LIN {X 0,Y 448.566,Z 349.616,A -85,B 0,C 180,E1 -8842.421,E2 -8842.421} C_VEL
LIN {X 0,Y 446.487,Z 338.496,A -85,B 0,C 180,E1 -8844.517,E2 -8844.517} C_VEL
LIN {X 0,Y 446.478,Z 338.493,A -85,B 0,C 180,E1 -8847.161,E2 -8847.161} C_VEL
LIN {X 0,Y 446.433,Z 338.501,A -85,B 0,C 180,E1 -8850.249,E2 -8850.249} C_VEL
LIN {X 0,Y 446.451,Z 338.496,A -85,B 0,C 180,E1 -8853.453,E2 -8853.453} C_VEL
LIN {X 0,Y 446.405,Z 338.501,A -85,B 0,C 180,E1 -8856.745,E2 -8856.745} C_VEL
LIN {X 0,Y 446.406,Z 338.503,A -85,B 0,C 180,E1 -8859.516,E2 -8859.516} C_VEL
LIN {X 0,Y 446.421,Z 338.499,A -85,B 0,C 180,E1 -8862.606,E2 -8862.606} C_VEL
LIN {X 0,Y 446.455,Z 338.496,A -85,B 0,C 180,E1 -8865.103,E2 -8865.103} C_VEL
LIN {X 0,Y 446.411,Z 338.5,A -85,B 0,C 180,E1 -8868.606,E2 -8868.606} C_VEL
LIN {X 0,Y 446.404,Z 338.505,A -85,B 0,C 180,E1 -8871.923,E2 -8871.923} C_VEL
LIN {X 0,Y 446.425,Z 338.501,A -85,B 0,C 180,E1 -8875.475,E2 -8875.475} C_VEL
LIN {X 0,Y 446.394,Z 338.506,A -85,B 0,C 180,E1 -8878.697,E2 -8878.697} C_VEL
LIN {X 0,Y 446.41,Z 338.504,A -85,B 0,C 180,E1 -8881.84,E2 -8881.84} C_VEL
LIN {X 0,Y 446.427,Z 338.66,A -85,B 0,C 180,E1 -8883.514,E2 -8883.514} C_VEL
LIN {X 0,Y 449.208,Z 351.748,A -85,B 0,C 180,E1 -8886.241,E2 -8886.241} C_VEL
LIN {X 0,Y 449.635,Z 355.585,A -85,B 0,C 180,E1 -8887.001,E2 -8887.001} C_VEL
LIN {X 0,Y 449.143,Z 363.301,A -85,B 0,C 180,E1 -8888.438,E2 -8888.438} C_VEL
LIN {X 0,Y 450.701,Z 371.004,A -85,B 0,C 180,E1 -8888.654,E2 -8888.654} C_VEL
LIN {X 0,Y 451.103,Z 376.824,A -85,B 0,C 180,E1 -8888.771,E2 -8888.771} C_VEL
LIN {X 0,Y 450.451,Z 382.718,A -85,B 0,C 180,E1 -8888.837,E2 -8888.837} C_VEL
LIN {X 0,Y 447.177,Z 398.482,A -85,B 0,C 180,E1 -8888.94,E2 -8888.94} C_VEL
LIN {X 0,Y 446.777,Z 402.479,A -85,B 0,C 180,E1 -8888.988,E2 -8888.988} C_VEL
LIN {X 0,Y 445.528,Z 498.742,A -85,B 0,C 180,E1 -8890.563,E2 -8890.563} C_VEL
LIN {X 0,Y 445.071,Z 513.383,A -85,B 0,C 180,E1 -8890.962,E2 -8890.962} C_VEL
LIN {X 0,Y 444.548,Z 526.67,A -85,B 0,C 180,E1 -8891.507,E2 -8891.507} C_VEL
LIN {X 0,Y 443.844,Z 539.571,A -85,B 0,C 180,E1 -8892.212,E2 -8892.212} C_VEL
LIN {X 0,Y 443.131,Z 551.657,A -85,B 0,C 180,E1 -8893.056,E2 -8893.056} C_VEL
LIN {X 0,Y 442.208,Z 563.631,A -85,B 0,C 180,E1 -8894.087,E2 -8894.087} C_VEL
LIN {X 0,Y 441.379,Z 574.55,A -85,B 0,C 180,E1 -8895.239,E2 -8895.239} C_VEL
LIN {X 0,Y 440.642,Z 584.036,A -85,B 0,C 180,E1 -8896.441,E2 -8896.441} C_VEL
LIN {X 0,Y 440.079,Z 592.855,A -85,B 0,C 180,E1 -8897.783,E2 -8897.783} C_VEL
LIN {X 0,Y 439.351,Z 601.602,A -85,B 0,C 180,E1 -8899.398,E2 -8899.398} C_VEL
LIN {X 0,Y 438.986,Z 607.768,A -85,B 0,C 180,E1 -8900.786,E2 -8900.786} C_VEL
LIN {X 0,Y 438.615,Z 614.306,A -85,B 0,C 180,E1 -8902.634,E2 -8902.634} C_VEL
LIN {X 0,Y 438.46,Z 619.203,A -85,B 0,C 180,E1 -8904.48,E2 -8904.48} C_VEL
LIN {X 0,Y 438.291,Z 622.617,A -85,B 0,C 180,E1 -8906.321,E2 -8906.321} C_VEL
LIN {X 0,Y 438.342,Z 623.801,A -85,B 0,C 180,E1 -8907.242,E2 -8907.242} C_VEL
LIN {X 0,Y 438.229,Z 625.165,A -85,B 0,C 180,E1 -8909.08,E2 -8909.08} C_VEL
LIN {X 0,Y 438.229,Z 625.204,A -85,B 0,C 180,E1 -8910.918,E2 -8910.918} C_VEL
LIN {X 0,Y 438.34,Z 623.919,A -85,B 0,C 180,E1 -8912.756,E2 -8912.756} C_VEL
LIN {X 0,Y 438.35,Z 621.277,A -85,B 0,C 180,E1 -8914.597,E2 -8914.597} C_VEL
LIN {X 0,Y 438.505,Z 617.205,A -85,B 0,C 180,E1 -8916.44,E2 -8916.44} C_VEL
LIN {X 0,Y 438.771,Z 611.583,A -85,B 0,C 180,E1 -8918.287,E2 -8918.287} C_VEL
LIN {X 0,Y 439.168,Z 605.239,A -85,B 0,C 180,E1 -8919.904,E2 -8919.904} C_VEL
LIN {X 0,Y 439.724,Z 597.348,A -85,B 0,C 180,E1 -8921.523,E2 -8921.523} C_VEL
LIN {X 0,Y 440.33,Z 588.346,A -85,B 0,C 180,E1 -8923.029,E2 -8923.029} C_VEL
LIN {X 0,Y 441.022,Z 579.149,A -85,B 0,C 180,E1 -8924.299,E2 -8924.299} C_VEL
LIN {X 0,Y 441.871,Z 568.079,A -85,B 0,C 180,E1 -8925.567,E2 -8925.567} C_VEL
LIN {X 0,Y 442.7,Z 557.061,A -85,B 0,C 180,E1 -8926.602,E2 -8926.602} C_VEL
LIN {X 0,Y 443.617,Z 543.849,A -85,B 0,C 180,E1 -8927.602,E2 -8927.602} C_VEL
LIN {X 0,Y 444.29,Z 531.223,A -85,B 0,C 180,E1 -8928.357,E2 -8928.357} C_VEL
LIN {X 0,Y 444.92,Z 517.384,A -85,B 0,C 180,E1 -8928.982,E2 -8928.982} C_VEL
LIN {X 0,Y 445.448,Z 502.754,A -85,B 0,C 180,E1 -8929.437,E2 -8929.437} C_VEL
LIN {X 0,Y 445.804,Z 478.658,A -85,B 0,C 180,E1 -8929.871,E2 -8929.871} C_VEL
LIN {X 0,Y 446.948,Z 386.866,A -85,B 0,C 180,E1 -8931.362,E2 -8931.362} C_VEL
LIN {X 0,Y 443.134,Z 367.334,A -85,B 0,C 180,E1 -8931.889,E2 -8931.889} C_VEL
LIN {X 0,Y 442.319,Z 363.353,A -85,B 0,C 180,E1 -8932.01,E2 -8932.01} C_VEL
LIN {X 0,Y 442.779,Z 356.138,A -85,B 0,C 180,E1 -8933.377,E2 -8933.377} C_VEL
LIN {X 0,Y 440.804,Z 345.968,A -85,B 0,C 180,E1 -8935.496,E2 -8935.496} C_VEL
LIN {X 0,Y 439.369,Z 339.384,A -85,B 0,C 180,E1 -8936.927,E2 -8936.927} C_VEL
LIN {X 0,Y 439.367,Z 339.383,A -85,B 0,C 180,E1 -8940.257,E2 -8940.257} C_VEL
LIN {X 0,Y 439.389,Z 339.379,A -85,B 0,C 180,E1 -8943.722,E2 -8943.722} C_VEL
LIN {X 0,Y 439.337,Z 339.389,A -85,B 0,C 180,E1 -8946.885,E2 -8946.885} C_VEL
LIN {X 0,Y 439.337,Z 339.382,A -85,B 0,C 180,E1 -8949.839,E2 -8949.839} C_VEL
LIN {X 0,Y 439.323,Z 339.387,A -85,B 0,C 180,E1 -8952.618,E2 -8952.618} C_VEL
LIN {X 0,Y 439.387,Z 339.377,A -85,B 0,C 180,E1 -8955.269,E2 -8955.269} C_VEL
LIN {X 0,Y 439.344,Z 339.386,A -85,B 0,C 180,E1 -8959.015,E2 -8959.015} C_VEL
LIN {X 0,Y 439.333,Z 339.378,A -85,B 0,C 180,E1 -8962.563,E2 -8962.563} C_VEL
LIN {X 0,Y 439.383,Z 339.381,A -85,B 0,C 180,E1 -8964.842,E2 -8964.842} C_VEL
LIN {X 0,Y 439.353,Z 339.372,A -85,B 0,C 180,E1 -8968.138,E2 -8968.138} C_VEL
LIN {X 0,Y 439.386,Z 339.372,A -85,B 0,C 180,E1 -8971.605,E2 -8971.605} C_VEL
LIN {X 0,Y 439.356,Z 339.37,A -85,B 0,C 180,E1 -8974.412,E2 -8974.412} C_VEL
LIN {X 0,Y 439.349,Z 339.38,A -85,B 0,C 180,E1 -8977.424,E2 -8977.424} C_VEL
LIN {X 0,Y 439.427,Z 339.36,A -85,B 0,C 180,E1 -8980.663,E2 -8980.663} C_VEL
LIN {X 0,Y 439.439,Z 339.369,A -85,B 0,C 180,E1 -8984.224,E2 -8984.224} C_VEL
LIN {X 0,Y 439.467,Z 339.364,A -85,B 0,C 180,E1 -8988.001,E2 -8988.001} C_VEL
LIN {X 0,Y 439.487,Z 339.359,A -85,B 0,C 180,E1 -8991.725,E2 -8991.725} C_VEL
LIN {X 0,Y 439.575,Z 339.355,A -85,B 0,C 180,E1 -8994.495,E2 -8994.495} C_VEL
LIN {X 0,Y 439.615,Z 339.349,A -85,B 0,C 180,E1 -8998.168,E2 -8998.168} C_VEL
LIN {X 0,Y 439.58,Z 339.354,A -85,B 0,C 180,E1 -9000.916,E2 -9000.916} C_VEL
LIN {X 0,Y 439.594,Z 339.352,A -85,B 0,C 180,E1 -9002.749,E2 -9002.749} C_VEL
LIN {X 0,Y 439.546,Z 339.361,A -85,B 0,C 180,E1 -9006.426,E2 -9006.426} C_VEL
LIN {X 0,Y 439.459,Z 339.365,A -85,B 0,C 180,E1 -9009.202,E2 -9009.202} C_VEL
LIN {X 0,Y 439.45,Z 339.367,A -85,B 0,C 180,E1 -9012.938,E2 -9012.938} C_VEL
LIN {X 0,Y 439.431,Z 339.373,A -85,B 0,C 180,E1 -9016.348,E2 -9016.348} C_VEL
LIN {X 0,Y 439.387,Z 339.374,A -85,B 0,C 180,E1 -9019.627,E2 -9019.627} C_VEL
LIN {X 0,Y 439.347,Z 339.372,A -85,B 0,C 180,E1 -9022.576,E2 -9022.576} C_VEL
LIN {X 0,Y 439.35,Z 339.379,A -85,B 0,C 180,E1 -9025.588,E2 -9025.588} C_VEL
LIN {X 0,Y 439.376,Z 339.369,A -85,B 0,C 180,E1 -9028.676,E2 -9028.676} C_VEL
LIN {X 0,Y 439.349,Z 339.383,A -85,B 0,C 180,E1 -9032.03,E2 -9032.03} C_VEL
LIN {X 0,Y 439.373,Z 339.376,A -85,B 0,C 180,E1 -9035.34,E2 -9035.34} C_VEL
LIN {X 0,Y 439.338,Z 339.385,A -85,B 0,C 180,E1 -9038.6,E2 -9038.6} C_VEL
LIN {X 0,Y 439.347,Z 339.379,A -85,B 0,C 180,E1 -9041.253,E2 -9041.253} C_VEL
LIN {X 0,Y 439.363,Z 339.381,A -85,B 0,C 180,E1 -9044.734,E2 -9044.734} C_VEL
LIN {X 0,Y 439.334,Z 339.386,A -85,B 0,C 180,E1 -9047.791,E2 -9047.791} C_VEL
LIN {X 0,Y 439.339,Z 339.383,A -85,B 0,C 180,E1 -9051.403,E2 -9051.403} C_VEL
LIN {X 0,Y 439.382,Z 339.378,A -85,B 0,C 180,E1 -9054.845,E2 -9054.845} C_VEL
LIN {X 0,Y 439.358,Z 339.383,A -85,B 0,C 180,E1 -9058.14,E2 -9058.14} C_VEL
LIN {X 0,Y 439.38,Z 339.378,A -85,B 0,C 180,E1 -9061.611,E2 -9061.611} C_VEL
LIN {X 0,Y 439.386,Z 339.457,A -85,B 0,C 180,E1 -9061.961,E2 -9061.961} C_VEL
LIN {X 0,Y 442.5,Z 353.697,A -85,B 0,C 180,E1 -9064.864,E2 -9064.864} C_VEL
LIN {X 0,Y 443.085,Z 357.713,A -85,B 0,C 180,E1 -9065.646,E2 -9065.646} C_VEL
LIN {X 0,Y 442.195,Z 370.912,A -85,B 0,C 180,E1 -9068.034,E2 -9068.034} C_VEL
LIN {X 0,Y 446.887,Z 395.742,A -85,B 0,C 180,E1 -9068.697,E2 -9068.697} C_VEL
LIN {X 0,Y 445.457,Z 507.784,A -85,B 0,C 180,E1 -9070.533,E2 -9070.533} C_VEL
LIN {X 0,Y 444.963,Z 521.924,A -85,B 0,C 180,E1 -9070.93,E2 -9070.93} C_VEL
LIN {X 0,Y 444.358,Z 535.626,A -85,B 0,C 180,E1 -9071.501,E2 -9071.501} C_VEL
LIN {X 0,Y 443.601,Z 549.079,A -85,B 0,C 180,E1 -9072.255,E2 -9072.255} C_VEL
LIN {X 0,Y 442.82,Z 561.734,A -85,B 0,C 180,E1 -9073.165,E2 -9073.165} C_VEL
LIN {X 0,Y 441.889,Z 573.37,A -85,B 0,C 180,E1 -9074.197,E2 -9074.197} C_VEL
LIN {X 0,Y 441.181,Z 583.057,A -85,B 0,C 180,E1 -9075.235,E2 -9075.235} C_VEL
LIN {X 0,Y 440.395,Z 593.68,A -85,B 0,C 180,E1 -9076.606,E2 -9076.606} C_VEL
LIN {X 0,Y 439.801,Z 602.653,A -85,B 0,C 180,E1 -9078.012,E2 -9078.012} C_VEL
LIN {X 0,Y 439.143,Z 611.145,A -85,B 0,C 180,E1 -9079.629,E2 -9079.629} C_VEL
LIN {X 0,Y 438.778,Z 617.986,A -85,B 0,C 180,E1 -9081.249,E2 -9081.249} C_VEL
LIN {X 0,Y 438.515,Z 622.7,A -85,B 0,C 180,E1 -9082.635,E2 -9082.635} C_VEL
LIN {X 0,Y 438.423,Z 627.591,A -85,B 0,C 180,E1 -9084.482,E2 -9084.482} C_VEL
LIN {X 0,Y 438.25,Z 630.988,A -85,B 0,C 180,E1 -9086.324,E2 -9086.324} C_VEL
LIN {X 0,Y 438.27,Z 632.994,A -85,B 0,C 180,E1 -9088.164,E2 -9088.164} C_VEL
LIN {X 0,Y 438.227,Z 633.656,A -85,B 0,C 180,E1 -9090.001,E2 -9090.001} C_VEL
LIN {X 0,Y 438.271,Z 632.988,A -85,B 0,C 180,E1 -9091.839,E2 -9091.839} C_VEL
LIN {X 0,Y 438.25,Z 630.975,A -85,B 0,C 180,E1 -9093.679,E2 -9093.679} C_VEL
LIN {X 0,Y 438.396,Z 627.576,A -85,B 0,C 180,E1 -9095.521,E2 -9095.521} C_VEL
LIN {X 0,Y 438.517,Z 622.686,A -85,B 0,C 180,E1 -9097.368,E2 -9097.368} C_VEL
LIN {X 0,Y 438.87,Z 616.152,A -85,B 0,C 180,E1 -9099.216,E2 -9099.216} C_VEL
LIN {X 0,Y 439.301,Z 608.881,A -85,B 0,C 180,E1 -9100.836,E2 -9100.836} C_VEL
LIN {X 0,Y 440.002,Z 599.879,A -85,B 0,C 180,E1 -9102.454,E2 -9102.454} C_VEL
LIN {X 0,Y 440.623,Z 590.428,A -85,B 0,C 180,E1 -9103.844,E2 -9103.844} C_VEL
LIN {X 0,Y 441.423,Z 579.967,A -85,B 0,C 180,E1 -9105.113,E2 -9105.113} C_VEL
LIN {X 0,Y 442.283,Z 568.419,A -85,B 0,C 180,E1 -9106.265,E2 -9106.265} C_VEL
LIN {X 0,Y 443.191,Z 555.607,A -85,B 0,C 180,E1 -9107.299,E2 -9107.299} C_VEL
LIN {X 0,Y 444.049,Z 542.285,A -85,B 0,C 180,E1 -9108.146,E2 -9108.146} C_VEL
LIN {X 0,Y 444.642,Z 529.175,A -85,B 0,C 180,E1 -9108.788,E2 -9108.788} C_VEL
LIN {X 0,Y 445.256,Z 515.429,A -85,B 0,C 180,E1 -9109.269,E2 -9109.269} C_VEL
LIN {X 0,Y 445.561,Z 501.404,A -85,B 0,C 180,E1 -9109.585,E2 -9109.585} C_VEL
LIN {X 0,Y 446.869,Z 395.827,A -85,B 0,C 180,E1 -9111.298,E2 -9111.298} C_VEL
LIN {X 0,Y 442.566,Z 372.827,A -85,B 0,C 180,E1 -9111.908,E2 -9111.908} C_VEL
LIN {X 0,Y 442.209,Z 370.731,A -85,B 0,C 180,E1 -9111.994,E2 -9111.994} C_VEL
LIN {X 0,Y 443.057,Z 357.667,A -85,B 0,C 180,E1 -9114.358,E2 -9114.358} C_VEL
LIN {X 0,Y 441.922,Z 350.934,A -85,B 0,C 180,E1 -9115.682,E2 -9115.682} C_VEL
LIN {X 0,Y 439.383,Z 339.381,A -85,B 0,C 180,E1 -9118.071,E2 -9118.071} C_VEL
LIN {X 0,Y 439.364,Z 339.382,A -85,B 0,C 180,E1 -9120.789,E2 -9120.789} C_VEL
LIN {X 0,Y 439.392,Z 339.377,A -85,B 0,C 180,E1 -9124.044,E2 -9124.044} C_VEL
LIN {X 0,Y 439.351,Z 339.381,A -85,B 0,C 180,E1 -9126.887,E2 -9126.887} C_VEL
LIN {X 0,Y 439.407,Z 339.372,A -85,B 0,C 180,E1 -9129.85,E2 -9129.85} C_VEL
LIN {X 0,Y 439.387,Z 339.377,A -85,B 0,C 180,E1 -9132.628,E2 -9132.628} C_VEL
LIN {X 0,Y 439.407,Z 339.376,A -85,B 0,C 180,E1 -9135.271,E2 -9135.271} C_VEL
LIN {X 0,Y 439.394,Z 339.378,A -85,B 0,C 180,E1 -9138.744,E2 -9138.744} C_VEL
LIN {X 0,Y 439.381,Z 339.377,A -85,B 0,C 180,E1 -9141.608,E2 -9141.608} C_VEL
LIN {X 0,Y 439.403,Z 339.375,A -85,B 0,C 180,E1 -9144.844,E2 -9144.844} C_VEL
LIN {X 0,Y 439.378,Z 339.382,A -85,B 0,C 180,E1 -9148.14,E2 -9148.14} C_VEL
LIN {X 0,Y 439.413,Z 339.381,A -85,B 0,C 180,E1 -9151.604,E2 -9151.604} C_VEL
LIN {X 0,Y 439.396,Z 339.439,A -85,B 0,C 180,E1 -9154.542,E2 -9154.542} C_VEL
LIN {X 0,Y 442.118,Z 350.97,A -85,B 0,C 180,E1 -9156.77,E2 -9156.77} C_VEL
LIN {X 0,Y 442.617,Z 355.527,A -85,B 0,C 180,E1 -9157.599,E2 -9157.599} C_VEL
LIN {X 0,Y 442.149,Z 372.27,A -85,B 0,C 180,E1 -9160.501,E2 -9160.501} C_VEL
LIN {X 0,Y 441.97,Z 378.87,A -85,B 0,C 180,E1 -9161.636,E2 -9161.636} C_VEL
LIN {X 0,Y 444.896,Z 393.264,A -85,B 0,C 180,E1 -9162.133,E2 -9162.133} C_VEL
LIN {X 0,Y 443.215,Z 477.735,A -85,B 0,C 180,E1 -9163.86,E2 -9163.86} C_VEL
LIN {X 0,Y 442.985,Z 491.998,A -85,B 0,C 180,E1 -9164.206,E2 -9164.206} C_VEL
LIN {X 0,Y 442.582,Z 504.819,A -85,B 0,C 180,E1 -9164.693,E2 -9164.693} C_VEL
LIN {X 0,Y 442.177,Z 515.784,A -85,B 0,C 180,E1 -9165.268,E2 -9165.268} C_VEL
LIN {X 0,Y 441.569,Z 528.484,A -85,B 0,C 180,E1 -9166.14,E2 -9166.14} C_VEL
LIN {X 0,Y 441.069,Z 539.531,A -85,B 0,C 180,E1 -9167.11,E2 -9167.11} C_VEL
LIN {X 0,Y 440.43,Z 550.006,A -85,B 0,C 180,E1 -9168.261,E2 -9168.261} C_VEL
LIN {X 0,Y 439.96,Z 558.544,A -85,B 0,C 180,E1 -9169.415,E2 -9169.415} C_VEL
LIN {X 0,Y 439.464,Z 566.835,A -85,B 0,C 180,E1 -9170.798,E2 -9170.798} C_VEL
LIN {X 0,Y 439.078,Z 573.477,A -85,B 0,C 180,E1 -9172.181,E2 -9172.181} C_VEL
LIN {X 0,Y 438.888,Z 578.742,A -85,B 0,C 180,E1 -9173.564,E2 -9173.564} C_VEL
LIN {X 0,Y 438.541,Z 582.812,A -85,B 0,C 180,E1 -9174.943,E2 -9174.943} C_VEL
LIN {X 0,Y 438.57,Z 585.775,A -85,B 0,C 180,E1 -9176.325,E2 -9176.325} C_VEL
LIN {X 0,Y 438.45,Z 587.197,A -85,B 0,C 180,E1 -9177.244,E2 -9177.244} C_VEL
LIN {X 0,Y 438.376,Z 588.173,A -85,B 0,C 180,E1 -9178.163,E2 -9178.163} C_VEL
LIN {X 0,Y 438.339,Z 588.748,A -85,B 0,C 180,E1 -9179.081,E2 -9179.081} C_VEL
LIN {X 0,Y 438.313,Z 588.9,A -85,B 0,C 180,E1 -9180,E2 -9180} C_VEL
LIN {X 0,Y 438.31,Z 588.599,A -85,B 0,C 180,E1 -9180.919,E2 -9180.919} C_VEL
LIN {X 0,Y 438.35,Z 587.898,A -85,B 0,C 180,E1 -9181.838,E2 -9181.838} C_VEL
LIN {X 0,Y 438.434,Z 586.788,A -85,B 0,C 180,E1 -9182.756,E2 -9182.756} C_VEL
LIN {X 0,Y 438.488,Z 584.28,A -85,B 0,C 180,E1 -9184.136,E2 -9184.136} C_VEL
LIN {X 0,Y 438.609,Z 580.731,A -85,B 0,C 180,E1 -9185.517,E2 -9185.517} C_VEL
LIN {X 0,Y 438.805,Z 575.437,A -85,B 0,C 180,E1 -9187.05,E2 -9187.05} C_VEL
LIN {X 0,Y 439.08,Z 568.932,A -85,B 0,C 180,E1 -9188.514,E2 -9188.514} C_VEL
LIN {X 0,Y 439.476,Z 561.185,A -85,B 0,C 180,E1 -9189.899,E2 -9189.899} C_VEL
LIN {X 0,Y 439.947,Z 551.471,A -85,B 0,C 180,E1 -9191.285,E2 -9191.285} C_VEL
LIN {X 0,Y 440.502,Z 541.396,A -85,B 0,C 180,E1 -9192.438,E2 -9192.438} C_VEL
LIN {X 0,Y 440.946,Z 530.681,A -85,B 0,C 180,E1 -9193.43,E2 -9193.43} C_VEL
LIN {X 0,Y 441.471,Z 519.08,A -85,B 0,C 180,E1 -9194.286,E2 -9194.286} C_VEL
LIN {X 0,Y 441.878,Z 506.81,A -85,B 0,C 180,E1 -9194.978,E2 -9194.978} C_VEL
LIN {X 0,Y 442.331,Z 493.591,A -85,B 0,C 180,E1 -9195.523,E2 -9195.523} C_VEL
LIN {X 0,Y 442.547,Z 480.562,A -85,B 0,C 180,E1 -9195.87,E2 -9195.87} C_VEL
LIN {X 0,Y 443.737,Z 392.63,A -85,B 0,C 180,E1 -9197.521,E2 -9197.521} C_VEL
LIN {X 0,Y 440.953,Z 376.477,A -85,B 0,C 180,E1 -9197.951,E2 -9197.951} C_VEL
LIN {X 0,Y 441.505,Z 358.045,A -85,B 0,C 180,E1 -9201.232,E2 -9201.232} C_VEL
LIN {X 0,Y 441.535,Z 350.426,A -85,B 0,C 180,E1 -9202.6,E2 -9202.6} C_VEL
LIN {X 0,Y 439.461,Z 339.371,A -85,B 0,C 180,E1 -9204.727,E2 -9204.727} C_VEL
LIN {X 0,Y 439.446,Z 339.371,A -85,B 0,C 180,E1 -9207.632,E2 -9207.632} C_VEL
LIN {X 0,Y 439.367,Z 339.376,A -85,B 0,C 180,E1 -9210.788,E2 -9210.788} C_VEL
LIN {X 0,Y 439.393,Z 339.379,A -85,B 0,C 180,E1 -9214.043,E2 -9214.043} C_VEL
LIN {X 0,Y 439.352,Z 339.38,A -85,B 0,C 180,E1 -9216.886,E2 -9216.886} C_VEL
LIN {X 0,Y 439.353,Z 339.386,A -85,B 0,C 180,E1 -9219.84,E2 -9219.84} C_VEL
LIN {X 0,Y 439.375,Z 339.377,A -85,B 0,C 180,E1 -9222.625,E2 -9222.625} C_VEL
LIN {X 0,Y 439.403,Z 339.376,A -85,B 0,C 180,E1 -9225.27,E2 -9225.27} C_VEL
LIN {X 0,Y 439.362,Z 339.38,A -85,B 0,C 180,E1 -9229.016,E2 -9229.016} C_VEL
LIN {X 0,Y 439.342,Z 339.382,A -85,B 0,C 180,E1 -9232.563,E2 -9232.563} C_VEL
LIN {X 0,Y 439.398,Z 339.376,A -85,B 0,C 180,E1 -9234.843,E2 -9234.843} C_VEL
LIN {X 0,Y 439.35,Z 339.383,A -85,B 0,C 180,E1 -9238.137,E2 -9238.137} C_VEL
LIN {X 0,Y 439.384,Z 339.382,A -85,B 0,C 180,E1 -9241.323,E2 -9241.323} C_VEL
LIN {X 0,Y 439.357,Z 339.437,A -85,B 0,C 180,E1 -9243.198,E2 -9243.198} C_VEL
LIN {X 0,Y 442.298,Z 353.087,A -85,B 0,C 180,E1 -9246.096,E2 -9246.096} C_VEL
LIN {X 0,Y 442.73,Z 357.158,A -85,B 0,C 180,E1 -9246.913,E2 -9246.913} C_VEL
LIN {X 0,Y 442.302,Z 363.377,A -85,B 0,C 180,E1 -9248.088,E2 -9248.088} C_VEL
LIN {X 0,Y 446.951,Z 386.317,A -85,B 0,C 180,E1 -9248.724,E2 -9248.724} C_VEL
LIN {X 0,Y 446.777,Z 402.479,A -85,B 0,C 180,E1 -9248.988,E2 -9248.988} C_VEL
LIN {X 0,Y 445.959,Z 408.324,A -85,B 0,C 180,E1 -9249.046,E2 -9249.046} C_VEL
LIN {X 0,Y 440.489,Z 427.373,A -85,B 0,C 180,E1 -9249.098,E2 -9249.098} C_VEL
LIN {X 0,Y 439.78,Z 433.216,A -85,B 0,C 180,E1 -9249.163,E2 -9249.163} C_VEL
LIN {X 0,Y 438.804,Z 500.275,A -85,B 0,C 180,E1 -9250.284,E2 -9250.284} C_VEL
LIN {X 0,Y 438.287,Z 515.011,A -85,B 0,C 180,E1 -9250.716,E2 -9250.716} C_VEL
LIN {X 0,Y 437.748,Z 527.879,A -85,B 0,C 180,E1 -9251.269,E2 -9251.269} C_VEL
LIN {X 0,Y 436.984,Z 541.227,A -85,B 0,C 180,E1 -9252.032,E2 -9252.032} C_VEL
LIN {X 0,Y 436.234,Z 553.154,A -85,B 0,C 180,E1 -9252.9,E2 -9252.9} C_VEL
LIN {X 0,Y 435.276,Z 564.875,A -85,B 0,C 180,E1 -9253.947,E2 -9253.947} C_VEL
LIN {X 0,Y 434.294,Z 576.569,A -85,B 0,C 180,E1 -9255.233,E2 -9255.233} C_VEL
LIN {X 0,Y 433.505,Z 586.646,A -85,B 0,C 180,E1 -9256.588,E2 -9256.588} C_VEL
LIN {X 0,Y 432.885,Z 595.628,A -85,B 0,C 180,E1 -9258.052,E2 -9258.052} C_VEL
LIN {X 0,Y 432.254,Z 603.886,A -85,B 0,C 180,E1 -9259.696,E2 -9259.696} C_VEL
LIN {X 0,Y 431.837,Z 609.642,A -85,B 0,C 180,E1 -9261.105,E2 -9261.105} C_VEL
LIN {X 0,Y 431.545,Z 614.375,A -85,B 0,C 180,E1 -9262.513,E2 -9262.513} C_VEL
LIN {X 0,Y 431.381,Z 619.272,A -85,B 0,C 180,E1 -9264.389,E2 -9264.389} C_VEL
LIN {X 0,Y 431.197,Z 622.685,A -85,B 0,C 180,E1 -9266.261,E2 -9266.261} C_VEL
LIN {X 0,Y 431.202,Z 624.716,A -85,B 0,C 180,E1 -9268.131,E2 -9268.131} C_VEL
LIN {X 0,Y 431.143,Z 625.417,A -85,B 0,C 180,E1 -9269.999,E2 -9269.999} C_VEL
LIN {X 0,Y 431.201,Z 624.795,A -85,B 0,C 180,E1 -9271.867,E2 -9271.867} C_VEL
LIN {X 0,Y 431.196,Z 622.837,A -85,B 0,C 180,E1 -9273.737,E2 -9273.737} C_VEL
LIN {X 0,Y 431.38,Z 619.492,A -85,B 0,C 180,E1 -9275.608,E2 -9275.608} C_VEL
LIN {X 0,Y 431.541,Z 614.663,A -85,B 0,C 180,E1 -9277.485,E2 -9277.485} C_VEL
LIN {X 0,Y 431.945,Z 608.204,A -85,B 0,C 180,E1 -9279.362,E2 -9279.362} C_VEL
LIN {X 0,Y 432.399,Z 601.013,A -85,B 0,C 180,E1 -9281.008,E2 -9281.008} C_VEL
LIN {X 0,Y 433.075,Z 593.473,A -85,B 0,C 180,E1 -9282.415,E2 -9282.415} C_VEL
LIN {X 0,Y 433.748,Z 583.935,A -85,B 0,C 180,E1 -9283.898,E2 -9283.898} C_VEL
LIN {X 0,Y 434.607,Z 573.457,A -85,B 0,C 180,E1 -9285.233,E2 -9285.233} C_VEL
LIN {X 0,Y 435.51,Z 562.281,A -85,B 0,C 180,E1 -9286.402,E2 -9286.402} C_VEL
LIN {X 0,Y 436.462,Z 549.915,A -85,B 0,C 180,E1 -9287.45,E2 -9287.45} C_VEL
LIN {X 0,Y 437.224,Z 537.403,A -85,B 0,C 180,E1 -9288.302,E2 -9288.302} C_VEL
LIN {X 0,Y 437.952,Z 523.666,A -85,B 0,C 180,E1 -9289.022,E2 -9289.022} C_VEL
LIN {X 0,Y 438.544,Z 509.091,A -85,B 0,C 180,E1 -9289.573,E2 -9289.573} C_VEL
LIN {X 0,Y 438.986,Z 494.622,A -85,B 0,C 180,E1 -9289.918,E2 -9289.918} C_VEL
LIN {X 0,Y 440.33,Z 387.141,A -85,B 0,C 180,E1 -9291.695,E2 -9291.695} C_VEL
LIN {X 0,Y 435.477,Z 363.381,A -85,B 0,C 180,E1 -9292.382,E2 -9292.382} C_VEL
LIN {X 0,Y 435.821,Z 358.176,A -85,B 0,C 180,E1 -9293.384,E2 -9293.384} C_VEL
LIN {X 0,Y 434.965,Z 352.386,A -85,B 0,C 180,E1 -9294.584,E2 -9294.584} C_VEL
LIN {X 0,Y 432.322,Z 340.261,A -85,B 0,C 180,E1 -9297.238,E2 -9297.238} C_VEL
LIN {X 0,Y 432.335,Z 340.26,A -85,B 0,C 180,E1 -9300.507,E2 -9300.507} C_VEL
LIN {X 0,Y 432.351,Z 340.256,A -85,B 0,C 180,E1 -9304.001,E2 -9304.001} C_VEL
LIN {X 0,Y 432.311,Z 340.261,A -85,B 0,C 180,E1 -9307.195,E2 -9307.195} C_VEL
LIN {X 0,Y 432.279,Z 340.262,A -85,B 0,C 180,E1 -9310.17,E2 -9310.17} C_VEL
LIN {X 0,Y 432.293,Z 340.264,A -85,B 0,C 180,E1 -9313.061,E2 -9313.061} C_VEL
LIN {X 0,Y 432.323,Z 340.255,A -85,B 0,C 180,E1 -9315.663,E2 -9315.663} C_VEL
LIN {X 0,Y 432.298,Z 340.26,A -85,B 0,C 180,E1 -9318.4,E2 -9318.4} C_VEL
LIN {X 0,Y 432.318,Z 340.248,A -85,B 0,C 180,E1 -9321.848,E2 -9321.848} C_VEL
LIN {X 0,Y 432.315,Z 340.255,A -85,B 0,C 180,E1 -9325.32,E2 -9325.32} C_VEL
LIN {X 0,Y 432.303,Z 340.255,A -85,B 0,C 180,E1 -9328.652,E2 -9328.652} C_VEL
LIN {X 0,Y 432.314,Z 340.253,A -85,B 0,C 180,E1 -9331.872,E2 -9331.872} C_VEL
LIN {X 0,Y 432.339,Z 340.251,A -85,B 0,C 180,E1 -9335.545,E2 -9335.545} C_VEL
LIN {X 0,Y 432.335,Z 340.248,A -85,B 0,C 180,E1 -9339.045,E2 -9339.045} C_VEL
LIN {X 0,Y 432.343,Z 340.242,A -85,B 0,C 180,E1 -9342.01,E2 -9342.01} C_VEL
LIN {X 0,Y 432.371,Z 340.252,A -85,B 0,C 180,E1 -9344.925,E2 -9344.925} C_VEL
LIN {X 0,Y 432.443,Z 340.238,A -85,B 0,C 180,E1 -9347.803,E2 -9347.803} C_VEL
LIN {X 0,Y 432.448,Z 340.236,A -85,B 0,C 180,E1 -9351.589,E2 -9351.589} C_VEL
LIN {X 0,Y 432.53,Z 340.234,A -85,B 0,C 180,E1 -9354.405,E2 -9354.405} C_VEL
LIN {X 0,Y 432.584,Z 340.225,A -85,B 0,C 180,E1 -9358.138,E2 -9358.138} C_VEL
LIN {X 0,Y 432.54,Z 340.23,A -85,B 0,C 180,E1 -9360.931,E2 -9360.931} C_VEL
LIN {X 0,Y 432.547,Z 340.229,A -85,B 0,C 180,E1 -9362.794,E2 -9362.794} C_VEL
LIN {X 0,Y 432.56,Z 340.224,A -85,B 0,C 180,E1 -9365.594,E2 -9365.594} C_VEL
LIN {X 0,Y 432.43,Z 340.243,A -85,B 0,C 180,E1 -9368.411,E2 -9368.411} C_VEL
LIN {X 0,Y 432.438,Z 340.244,A -85,B 0,C 180,E1 -9372.197,E2 -9372.197} C_VEL
LIN {X 0,Y 432.415,Z 340.245,A -85,B 0,C 180,E1 -9376.039,E2 -9376.039} C_VEL
LIN {X 0,Y 432.372,Z 340.248,A -85,B 0,C 180,E1 -9379.485,E2 -9379.485} C_VEL
LIN {X 0,Y 432.295,Z 340.252,A -85,B 0,C 180,E1 -9382.966,E2 -9382.966} C_VEL
LIN {X 0,Y 432.303,Z 340.26,A -85,B 0,C 180,E1 -9386.036,E2 -9386.036} C_VEL
LIN {X 0,Y 432.312,Z 340.247,A -85,B 0,C 180,E1 -9389.19,E2 -9389.19} C_VEL
LIN {X 0,Y 432.307,Z 340.26,A -85,B 0,C 180,E1 -9392.444,E2 -9392.444} C_VEL
LIN {X 0,Y 432.319,Z 340.257,A -85,B 0,C 180,E1 -9395.82,E2 -9395.82} C_VEL
LIN {X 0,Y 432.286,Z 340.26,A -85,B 0,C 180,E1 -9399.35,E2 -9399.35} C_VEL
LIN {X 0,Y 432.288,Z 340.26,A -85,B 0,C 180,E1 -9401.802,E2 -9401.802} C_VEL
LIN {X 0,Y 432.321,Z 340.263,A -85,B 0,C 180,E1 -9404.349,E2 -9404.349} C_VEL
LIN {X 0,Y 432.29,Z 340.261,A -85,B 0,C 180,E1 -9407.02,E2 -9407.02} C_VEL
LIN {X 0,Y 432.277,Z 340.266,A -85,B 0,C 180,E1 -9409.83,E2 -9409.83} C_VEL
LIN {X 0,Y 432.286,Z 340.262,A -85,B 0,C 180,E1 -9413.022,E2 -9413.022} C_VEL
LIN {X 0,Y 432.324,Z 340.261,A -85,B 0,C 180,E1 -9416.004,E2 -9416.004} C_VEL
LIN {X 0,Y 432.334,Z 340.255,A -85,B 0,C 180,E1 -9419.493,E2 -9419.493} C_VEL
LIN {X 0,Y 432.377,Z 340.426,A -85,B 0,C 180,E1 -9421.668,E2 -9421.668} C_VEL
LIN {X 0,Y 435.506,Z 354.776,A -85,B 0,C 180,E1 -9424.649,E2 -9424.649} C_VEL
LIN {X 0,Y 436.202,Z 358.993,A -85,B 0,C 180,E1 -9425.49,E2 -9425.49} C_VEL
LIN {X 0,Y 435.394,Z 370.89,A -85,B 0,C 180,E1 -9427.674,E2 -9427.674} C_VEL
LIN {X 0,Y 440.276,Z 396.519,A -85,B 0,C 180,E1 -9428.375,E2 -9428.375} C_VEL
LIN {X 0,Y 438.769,Z 507.731,A -85,B 0,C 180,E1 -9430.224,E2 -9430.224} C_VEL
LIN {X 0,Y 438.254,Z 521.864,A -85,B 0,C 180,E1 -9430.627,E2 -9430.627} C_VEL
LIN {X 0,Y 437.624,Z 535.564,A -85,B 0,C 180,E1 -9431.206,E2 -9431.206} C_VEL
LIN {X 0,Y 436.811,Z 549.336,A -85,B 0,C 180,E1 -9431.992,E2 -9431.992} C_VEL
LIN {X 0,Y 436.011,Z 561.67,A -85,B 0,C 180,E1 -9432.894,E2 -9432.894} C_VEL
LIN {X 0,Y 435.062,Z 573.305,A -85,B 0,C 180,E1 -9433.942,E2 -9433.942} C_VEL
LIN {X 0,Y 434.279,Z 582.992,A -85,B 0,C 180,E1 -9434.995,E2 -9434.995} C_VEL
LIN {X 0,Y 433.444,Z 593.729,A -85,B 0,C 180,E1 -9436.404,E2 -9436.404} C_VEL
LIN {X 0,Y 432.806,Z 602.587,A -85,B 0,C 180,E1 -9437.815,E2 -9437.815} C_VEL
LIN {X 0,Y 432.128,Z 611.079,A -85,B 0,C 180,E1 -9439.459,E2 -9439.459} C_VEL
LIN {X 0,Y 431.723,Z 617.919,A -85,B 0,C 180,E1 -9441.105,E2 -9441.105} C_VEL
LIN {X 0,Y 431.446,Z 622.634,A -85,B 0,C 180,E1 -9442.514,E2 -9442.514} C_VEL
LIN {X 0,Y 431.321,Z 627.524,A -85,B 0,C 180,E1 -9444.391,E2 -9444.391} C_VEL
LIN {X 0,Y 431.159,Z 630.921,A -85,B 0,C 180,E1 -9446.263,E2 -9446.263} C_VEL
LIN {X 0,Y 431.194,Z 632.927,A -85,B 0,C 180,E1 -9448.133,E2 -9448.133} C_VEL
LIN {X 0,Y 431.142,Z 633.589,A -85,B 0,C 180,E1 -9450.001,E2 -9450.001} C_VEL
LIN {X 0,Y 431.194,Z 632.921,A -85,B 0,C 180,E1 -9451.869,E2 -9451.869} C_VEL
LIN {X 0,Y 431.159,Z 630.908,A -85,B 0,C 180,E1 -9453.74,E2 -9453.74} C_VEL
LIN {X 0,Y 431.298,Z 627.508,A -85,B 0,C 180,E1 -9455.612,E2 -9455.612} C_VEL
LIN {X 0,Y 431.449,Z 622.617,A -85,B 0,C 180,E1 -9457.489,E2 -9457.489} C_VEL
LIN {X 0,Y 431.811,Z 616.084,A -85,B 0,C 180,E1 -9459.368,E2 -9459.368} C_VEL
LIN {X 0,Y 432.302,Z 608.812,A -85,B 0,C 180,E1 -9461.014,E2 -9461.014} C_VEL
LIN {X 0,Y 432.933,Z 601.194,A -85,B 0,C 180,E1 -9462.422,E2 -9462.422} C_VEL
LIN {X 0,Y 433.558,Z 592.214,A -85,B 0,C 180,E1 -9463.811,E2 -9463.811} C_VEL
LIN {X 0,Y 434.292,Z 582.937,A -85,B 0,C 180,E1 -9465.007,E2 -9465.007} C_VEL
LIN {X 0,Y 435.175,Z 572.063,A -85,B 0,C 180,E1 -9466.177,E2 -9466.177} C_VEL
LIN {X 0,Y 436.132,Z 560.156,A -85,B 0,C 180,E1 -9467.225,E2 -9467.225} C_VEL
LIN {X 0,Y 436.99,Z 547.963,A -85,B 0,C 180,E1 -9468.091,E2 -9468.091} C_VEL
LIN {X 0,Y 437.686,Z 534.289,A -85,B 0,C 180,E1 -9468.855,E2 -9468.855} C_VEL
LIN {X 0,Y 438.335,Z 520.847,A -85,B 0,C 180,E1 -9469.403,E2 -9469.403} C_VEL
LIN {X 0,Y 438.77,Z 507.375,A -85,B 0,C 180,E1 -9469.779,E2 -9469.779} C_VEL
LIN {X 0,Y 440.237,Z 396.801,A -85,B 0,C 180,E1 -9471.617,E2 -9471.617} C_VEL
LIN {X 0,Y 436.376,Z 375.906,A -85,B 0,C 180,E1 -9472.18,E2 -9472.18} C_VEL
LIN {X 0,Y 435.4,Z 370.758,A -85,B 0,C 180,E1 -9472.338,E2 -9472.338} C_VEL
LIN {X 0,Y 436.178,Z 358.945,A -85,B 0,C 180,E1 -9474.514,E2 -9474.514} C_VEL
LIN {X 0,Y 434.393,Z 349.519,A -85,B 0,C 180,E1 -9476.419,E2 -9476.419} C_VEL
LIN {X 0,Y 432.358,Z 340.254,A -85,B 0,C 180,E1 -9478.378,E2 -9478.378} C_VEL
LIN {X 0,Y 432.325,Z 340.258,A -85,B 0,C 180,E1 -9481.347,E2 -9481.347} C_VEL
LIN {X 0,Y 432.344,Z 340.254,A -85,B 0,C 180,E1 -9484.678,E2 -9484.678} C_VEL
LIN {X 0,Y 432.34,Z 340.253,A -85,B 0,C 180,E1 -9488.151,E2 -9488.151} C_VEL
LIN {X 0,Y 432.338,Z 340.255,A -85,B 0,C 180,E1 -9491.603,E2 -9491.603} C_VEL
LIN {X 0,Y 432.339,Z 340.254,A -85,B 0,C 180,E1 -9494.348,E2 -9494.348} C_VEL
LIN {X 0,Y 432.326,Z 340.26,A -85,B 0,C 180,E1 -9497.016,E2 -9497.016} C_VEL
LIN {X 0,Y 432.338,Z 340.255,A -85,B 0,C 180,E1 -9499.821,E2 -9499.821} C_VEL
LIN {X 0,Y 432.31,Z 340.258,A -85,B 0,C 180,E1 -9503.022,E2 -9503.022} C_VEL
LIN {X 0,Y 432.364,Z 340.255,A -85,B 0,C 180,E1 -9505.997,E2 -9505.997} C_VEL
LIN {X 0,Y 432.351,Z 340.257,A -85,B 0,C 180,E1 -9509.49,E2 -9509.49} C_VEL
LIN {X 0,Y 432.351,Z 340.262,A -85,B 0,C 180,E1 -9511.875,E2 -9511.875} C_VEL
LIN {X 0,Y 432.359,Z 340.268,A -85,B 0,C 180,E1 -9514.097,E2 -9514.097} C_VEL
LIN {X 0,Y 434.981,Z 350.789,A -85,B 0,C 180,E1 -9516.176,E2 -9516.176} C_VEL
LIN {X 0,Y 435.888,Z 356.313,A -85,B 0,C 180,E1 -9517.234,E2 -9517.234} C_VEL
LIN {X 0,Y 435.425,Z 373.191,A -85,B 0,C 180,E1 -9520.187,E2 -9520.187} C_VEL
LIN {X 0,Y 435.214,Z 379.143,A -85,B 0,C 180,E1 -9521.232,E2 -9521.232} C_VEL
LIN {X 0,Y 438.339,Z 394.131,A -85,B 0,C 180,E1 -9521.786,E2 -9521.786} C_VEL
LIN {X 0,Y 436.531,Z 477.297,A -85,B 0,C 180,E1 -9523.546,E2 -9523.546} C_VEL
LIN {X 0,Y 436.278,Z 491.718,A -85,B 0,C 180,E1 -9523.896,E2 -9523.896} C_VEL
LIN {X 0,Y 435.848,Z 504.646,A -85,B 0,C 180,E1 -9524.39,E2 -9524.39} C_VEL
LIN {X 0,Y 435.369,Z 516.663,A -85,B 0,C 180,E1 -9525.032,E2 -9525.032} C_VEL
LIN {X 0,Y 434.702,Z 529.859,A -85,B 0,C 180,E1 -9525.965,E2 -9525.965} C_VEL
LIN {X 0,Y 434.105,Z 541.32,A -85,B 0,C 180,E1 -9527.019,E2 -9527.019} C_VEL
LIN {X 0,Y 433.508,Z 550.607,A -85,B 0,C 180,E1 -9528.071,E2 -9528.071} C_VEL
LIN {X 0,Y 433.01,Z 559.107,A -85,B 0,C 180,E1 -9529.243,E2 -9529.243} C_VEL
LIN {X 0,Y 432.491,Z 567.353,A -85,B 0,C 180,E1 -9530.648,E2 -9530.648} C_VEL
LIN {X 0,Y 432.063,Z 573.966,A -85,B 0,C 180,E1 -9532.053,E2 -9532.053} C_VEL
LIN {X 0,Y 431.85,Z 579.204,A -85,B 0,C 180,E1 -9533.459,E2 -9533.459} C_VEL
LIN {X 0,Y 431.48,Z 583.254,A -85,B 0,C 180,E1 -9534.86,E2 -9534.86} C_VEL
LIN {X 0,Y 431.511,Z 586.192,A -85,B 0,C 180,E1 -9536.265,E2 -9536.265} C_VEL
LIN {X 0,Y 431.383,Z 587.586,A -85,B 0,C 180,E1 -9537.199,E2 -9537.199} C_VEL
LIN {X 0,Y 431.297,Z 588.548,A -85,B 0,C 180,E1 -9538.132,E2 -9538.132} C_VEL
LIN {X 0,Y 431.252,Z 589.107,A -85,B 0,C 180,E1 -9539.066,E2 -9539.066} C_VEL
LIN {X 0,Y 431.224,Z 589.228,A -85,B 0,C 180,E1 -9540,E2 -9540} C_VEL
LIN {X 0,Y 431.225,Z 588.907,A -85,B 0,C 180,E1 -9540.934,E2 -9540.934} C_VEL
LIN {X 0,Y 431.272,Z 588.185,A -85,B 0,C 180,E1 -9541.868,E2 -9541.868} C_VEL
LIN {X 0,Y 431.365,Z 587.043,A -85,B 0,C 180,E1 -9542.802,E2 -9542.802} C_VEL
LIN {X 0,Y 431.395,Z 584.489,A -85,B 0,C 180,E1 -9544.204,E2 -9544.204} C_VEL
LIN {X 0,Y 431.539,Z 580.882,A -85,B 0,C 180,E1 -9545.608,E2 -9545.608} C_VEL
LIN {X 0,Y 431.73,Z 575.296,A -85,B 0,C 180,E1 -9547.224,E2 -9547.224} C_VEL
LIN {X 0,Y 432.032,Z 568.946,A -85,B 0,C 180,E1 -9548.654,E2 -9548.654} C_VEL
LIN {X 0,Y 432.451,Z 561.089,A -85,B 0,C 180,E1 -9550.062,E2 -9550.062} C_VEL
LIN {X 0,Y 432.935,Z 551.277,A -85,B 0,C 180,E1 -9551.47,E2 -9551.47} C_VEL
LIN {X 0,Y 433.544,Z 541.042,A -85,B 0,C 180,E1 -9552.641,E2 -9552.641} C_VEL
LIN {X 0,Y 434.025,Z 529.641,A -85,B 0,C 180,E1 -9553.695,E2 -9553.695} C_VEL
LIN {X 0,Y 434.525,Z 518.301,A -85,B 0,C 180,E1 -9554.519,E2 -9554.519} C_VEL
LIN {X 0,Y 434.999,Z 505.747,A -85,B 0,C 180,E1 -9555.221,E2 -9555.221} C_VEL
LIN {X 0,Y 435.41,Z 492.751,A -85,B 0,C 180,E1 -9555.746,E2 -9555.746} C_VEL
LIN {X 0,Y 435.631,Z 479.085,A -85,B 0,C 180,E1 -9556.098,E2 -9556.098} C_VEL
LIN {X 0,Y 436.889,Z 393.499,A -85,B 0,C 180,E1 -9557.742,E2 -9557.742} C_VEL
LIN {X 0,Y 434.007,Z 376.628,A -85,B 0,C 180,E1 -9558.214,E2 -9558.214} C_VEL
LIN {X 0,Y 434.629,Z 357.833,A -85,B 0,C 180,E1 -9561.584,E2 -9561.584} C_VEL
LIN {X 0,Y 434.509,Z 351.236,A -85,B 0,C 180,E1 -9562.785,E2 -9562.785} C_VEL
LIN {X 0,Y 432.393,Z 340.251,A -85,B 0,C 180,E1 -9564.893,E2 -9564.893} C_VEL
LIN {X 0,Y 432.388,Z 340.253,A -85,B 0,C 180,E1 -9568.123,E2 -9568.123} C_VEL
LIN {X 0,Y 432.327,Z 340.253,A -85,B 0,C 180,E1 -9571.346,E2 -9571.346} C_VEL
LIN {X 0,Y 432.345,Z 340.253,A -85,B 0,C 180,E1 -9574.677,E2 -9574.677} C_VEL
LIN {X 0,Y 432.335,Z 340.257,A -85,B 0,C 180,E1 -9578.15,E2 -9578.15} C_VEL
LIN {X 0,Y 432.326,Z 340.261,A -85,B 0,C 180,E1 -9581.798,E2 -9581.798} C_VEL
LIN {X 0,Y 432.339,Z 340.255,A -85,B 0,C 180,E1 -9584.347,E2 -9584.347} C_VEL
LIN {X 0,Y 432.312,Z 340.258,A -85,B 0,C 180,E1 -9587.017,E2 -9587.017} C_VEL
LIN {X 0,Y 432.294,Z 340.263,A -85,B 0,C 180,E1 -9589.827,E2 -9589.827} C_VEL
LIN {X 0,Y 432.303,Z 340.261,A -85,B 0,C 180,E1 -9593.02,E2 -9593.02} C_VEL
LIN {X 0,Y 432.337,Z 340.257,A -85,B 0,C 180,E1 -9596.001,E2 -9596.001} C_VEL
LIN {X 0,Y 432.342,Z 340.256,A -85,B 0,C 180,E1 -9599.491,E2 -9599.491} C_VEL
LIN {X 0,Y 432.317,Z 340.253,A -85,B 0,C 180,E1 -9602.857,E2 -9602.857} C_VEL
LIN {X 0,Y 435.36,Z 354.429,A -85,B 0,C 180,E1 -9605.944,E2 -9605.944} C_VEL
LIN {X 0,Y 435.833,Z 358.634,A -85,B 0,C 180,E1 -9606.803,E2 -9606.803} C_VEL
LIN {X 0,Y 435.466,Z 363.454,A -85,B 0,C 180,E1 -9607.727,E2 -9607.727} C_VEL
LIN {X 0,Y 440.377,Z 387.516,A -85,B 0,C 180,E1 -9608.409,E2 -9608.409} C_VEL
LIN {X 0,Y 439.78,Z 433.216,A -85,B 0,C 180,E1 -9609.163,E2 -9609.163} C_VEL
LIN {X 0,Y 439.041,Z 439.064,A -85,B 0,C 180,E1 -9609.226,E2 -9609.226} C_VEL
LIN {X 0,Y 433.479,Z 458.099,A -85,B 0,C 180,E1 -9609.277,E2 -9609.277} C_VEL
LIN {X 0,Y 432.788,Z 463.945,A -85,B 0,C 180,E1 -9609.344,E2 -9609.344} C_VEL
LIN {X 0,Y 432.088,Z 501.522,A -85,B 0,C 180,E1 -9609.995,E2 -9609.995} C_VEL
LIN {X 0,Y 431.571,Z 515.851,A -85,B 0,C 180,E1 -9610.435,E2 -9610.435} C_VEL
LIN {X 0,Y 430.933,Z 529.557,A -85,B 0,C 180,E1 -9611.05,E2 -9611.05} C_VEL
LIN {X 0,Y 430.146,Z 542.669,A -85,B 0,C 180,E1 -9611.832,E2 -9611.832} C_VEL
LIN {X 0,Y 429.339,Z 554.65,A -85,B 0,C 180,E1 -9612.74,E2 -9612.74} C_VEL
LIN {X 0,Y 428.314,Z 566.12,A -85,B 0,C 180,E1 -9613.802,E2 -9613.802} C_VEL
LIN {X 0,Y 427.43,Z 576.64,A -85,B 0,C 180,E1 -9614.99,E2 -9614.99} C_VEL
LIN {X 0,Y 426.537,Z 587.248,A -85,B 0,C 180,E1 -9616.444,E2 -9616.444} C_VEL
LIN {X 0,Y 425.907,Z 595.698,A -85,B 0,C 180,E1 -9617.853,E2 -9617.853} C_VEL
LIN {X 0,Y 425.208,Z 603.956,A -85,B 0,C 180,E1 -9619.523,E2 -9619.523} C_VEL
LIN {X 0,Y 424.81,Z 609.711,A -85,B 0,C 180,E1 -9620.956,E2 -9620.956} C_VEL
LIN {X 0,Y 424.501,Z 614.444,A -85,B 0,C 180,E1 -9622.388,E2 -9622.388} C_VEL
LIN {X 0,Y 424.289,Z 619.34,A -85,B 0,C 180,E1 -9624.295,E2 -9624.295} C_VEL
LIN {X 0,Y 424.108,Z 622.753,A -85,B 0,C 180,E1 -9626.198,E2 -9626.198} C_VEL
LIN {X 0,Y 424.128,Z 624.784,A -85,B 0,C 180,E1 -9628.099,E2 -9628.099} C_VEL
LIN {X 0,Y 424.061,Z 625.484,A -85,B 0,C 180,E1 -9629.999,E2 -9629.999} C_VEL
LIN {X 0,Y 424.127,Z 624.862,A -85,B 0,C 180,E1 -9631.898,E2 -9631.898} C_VEL
LIN {X 0,Y 424.107,Z 622.904,A -85,B 0,C 180,E1 -9633.799,E2 -9633.799} C_VEL
LIN {X 0,Y 424.286,Z 619.559,A -85,B 0,C 180,E1 -9635.702,E2 -9635.702} C_VEL
LIN {X 0,Y 424.497,Z 614.729,A -85,B 0,C 180,E1 -9637.61,E2 -9637.61} C_VEL
LIN {X 0,Y 424.909,Z 608.27,A -85,B 0,C 180,E1 -9639.519,E2 -9639.519} C_VEL
LIN {X 0,Y 425.387,Z 601.078,A -85,B 0,C 180,E1 -9641.192,E2 -9641.192} C_VEL
LIN {X 0,Y 426.119,Z 593.538,A -85,B 0,C 180,E1 -9642.621,E2 -9642.621} C_VEL
LIN {X 0,Y 426.784,Z 584.489,A -85,B 0,C 180,E1 -9644.055,E2 -9644.055} C_VEL
LIN {X 0,Y 427.745,Z 573.521,A -85,B 0,C 180,E1 -9645.484,E2 -9645.484} C_VEL
LIN {X 0,Y 428.69,Z 562.343,A -85,B 0,C 180,E1 -9646.671,E2 -9646.671} C_VEL
LIN {X 0,Y 429.662,Z 549.977,A -85,B 0,C 180,E1 -9647.735,E2 -9647.735} C_VEL
LIN {X 0,Y 430.513,Z 537.307,A -85,B 0,C 180,E1 -9648.607,E2 -9648.607} C_VEL
LIN {X 0,Y 431.242,Z 523.724,A -85,B 0,C 180,E1 -9649.33,E2 -9649.33} C_VEL
LIN {X 0,Y 431.861,Z 509.145,A -85,B 0,C 180,E1 -9649.889,E2 -9649.889} C_VEL
LIN {X 0,Y 432.327,Z 494.667,A -85,B 0,C 180,E1 -9650.238,E2 -9650.238} C_VEL
LIN {X 0,Y 433.749,Z 388.88,A -85,B 0,C 180,E1 -9652.011,E2 -9652.011} C_VEL
LIN {X 0,Y 429.014,Z 365.321,A -85,B 0,C 180,E1 -9652.686,E2 -9652.686} C_VEL
LIN {X 0,Y 428.627,Z 363.509,A -85,B 0,C 180,E1 -9652.747,E2 -9652.747} C_VEL
LIN {X 0,Y 428.88,Z 358.593,A -85,B 0,C 180,E1 -9653.715,E2 -9653.715} C_VEL
LIN {X 0,Y 426.673,Z 347.366,A -85,B 0,C 180,E1 -9656.141,E2 -9656.141} C_VEL
LIN {X 0,Y 425.272,Z 341.14,A -85,B 0,C 180,E1 -9657.561,E2 -9657.561} C_VEL
LIN {X 0,Y 425.28,Z 341.141,A -85,B 0,C 180,E1 -9660.815,E2 -9660.815} C_VEL
LIN {X 0,Y 425.303,Z 341.135,A -85,B 0,C 180,E1 -9664.286,E2 -9664.286} C_VEL
LIN {X 0,Y 425.266,Z 341.135,A -85,B 0,C 180,E1 -9667.693,E2 -9667.693} C_VEL
LIN {X 0,Y 425.234,Z 341.142,A -85,B 0,C 180,E1 -9670.513,E2 -9670.513} C_VEL
LIN {X 0,Y 425.236,Z 341.14,A -85,B 0,C 180,E1 -9673.348,E2 -9673.348} C_VEL
LIN {X 0,Y 425.247,Z 341.136,A -85,B 0,C 180,E1 -9676.042,E2 -9676.042} C_VEL
LIN {X 0,Y 425.238,Z 341.141,A -85,B 0,C 180,E1 -9678.617,E2 -9678.617} C_VEL
LIN {X 0,Y 425.269,Z 341.13,A -85,B 0,C 180,E1 -9681.098,E2 -9681.098} C_VEL
LIN {X 0,Y 425.283,Z 341.137,A -85,B 0,C 180,E1 -9684.662,E2 -9684.662} C_VEL
LIN {X 0,Y 425.248,Z 341.128,A -85,B 0,C 180,E1 -9688.071,E2 -9688.071} C_VEL
LIN {X 0,Y 425.291,Z 341.129,A -85,B 0,C 180,E1 -9691.365,E2 -9691.365} C_VEL
LIN {X 0,Y 425.247,Z 341.128,A -85,B 0,C 180,E1 -9694.551,E2 -9694.551} C_VEL
LIN {X 0,Y 425.278,Z 341.132,A -85,B 0,C 180,E1 -9697.729,E2 -9697.729} C_VEL
LIN {X 0,Y 425.347,Z 341.112,A -85,B 0,C 180,E1 -9700.703,E2 -9700.703} C_VEL
LIN {X 0,Y 425.371,Z 341.119,A -85,B 0,C 180,E1 -9703.687,E2 -9703.687} C_VEL
LIN {X 0,Y 425.397,Z 341.116,A -85,B 0,C 180,E1 -9707.598,E2 -9707.598} C_VEL
LIN {X 0,Y 425.392,Z 341.115,A -85,B 0,C 180,E1 -9711.449,E2 -9711.449} C_VEL
LIN {X 0,Y 425.488,Z 341.11,A -85,B 0,C 180,E1 -9714.312,E2 -9714.312} C_VEL
LIN {X 0,Y 425.553,Z 341.1,A -85,B 0,C 180,E1 -9718.107,E2 -9718.107} C_VEL
LIN {X 0,Y 425.502,Z 341.107,A -85,B 0,C 180,E1 -9720.946,E2 -9720.946} C_VEL
LIN {X 0,Y 425.502,Z 341.106,A -85,B 0,C 180,E1 -9722.84,E2 -9722.84} C_VEL
LIN {X 0,Y 425.514,Z 341.102,A -85,B 0,C 180,E1 -9725.687,E2 -9725.687} C_VEL
LIN {X 0,Y 425.379,Z 341.121,A -85,B 0,C 180,E1 -9728.551,E2 -9728.551} C_VEL
LIN {X 0,Y 425.393,Z 341.12,A -85,B 0,C 180,E1 -9732.402,E2 -9732.402} C_VEL
LIN {X 0,Y 425.372,Z 341.123,A -85,B 0,C 180,E1 -9736.312,E2 -9736.312} C_VEL
LIN {X 0,Y 425.314,Z 341.127,A -85,B 0,C 180,E1 -9739.636,E2 -9739.636} C_VEL
LIN {X 0,Y 425.273,Z 341.123,A -85,B 0,C 180,E1 -9742.34,E2 -9742.34} C_VEL
LIN {X 0,Y 425.244,Z 341.136,A -85,B 0,C 180,E1 -9745.449,E2 -9745.449} C_VEL
LIN {X 0,Y 425.293,Z 341.122,A -85,B 0,C 180,E1 -9748.861,E2 -9748.861} C_VEL
LIN {X 0,Y 425.247,Z 341.139,A -85,B 0,C 180,E1 -9751.928,E2 -9751.928} C_VEL
LIN {X 0,Y 425.279,Z 341.132,A -85,B 0,C 180,E1 -9755.338,E2 -9755.338} C_VEL
LIN {X 0,Y 425.261,Z 341.136,A -85,B 0,C 180,E1 -9758.903,E2 -9758.903} C_VEL
LIN {X 0,Y 425.242,Z 341.14,A -85,B 0,C 180,E1 -9762.657,E2 -9762.657} C_VEL
LIN {X 0,Y 425.272,Z 341.134,A -85,B 0,C 180,E1 -9765.285,E2 -9765.285} C_VEL
LIN {X 0,Y 425.234,Z 341.143,A -85,B 0,C 180,E1 -9768.619,E2 -9768.619} C_VEL
LIN {X 0,Y 425.259,Z 341.142,A -85,B 0,C 180,E1 -9772.306,E2 -9772.306} C_VEL
LIN {X 0,Y 425.277,Z 341.138,A -85,B 0,C 180,E1 -9775.817,E2 -9775.817} C_VEL
LIN {X 0,Y 425.282,Z 341.133,A -85,B 0,C 180,E1 -9779.241,E2 -9779.241} C_VEL
LIN {X 0,Y 425.302,Z 341.272,A -85,B 0,C 180,E1 -9781.335,E2 -9781.335} C_VEL
LIN {X 0,Y 427.999,Z 353.443,A -85,B 0,C 180,E1 -9783.926,E2 -9783.926} C_VEL
LIN {X 0,Y 429.321,Z 360.272,A -85,B 0,C 180,E1 -9785.329,E2 -9785.329} C_VEL
LIN {X 0,Y 428.557,Z 370.712,A -85,B 0,C 180,E1 -9787.284,E2 -9787.284} C_VEL
LIN {X 0,Y 433.62,Z 396.813,A -85,B 0,C 180,E1 -9788.032,E2 -9788.032} C_VEL
LIN {X 0,Y 432.114,Z 507.679,A -85,B 0,C 180,E1 -9789.907,E2 -9789.907} C_VEL
LIN {X 0,Y 431.58,Z 521.805,A -85,B 0,C 180,E1 -9790.315,E2 -9790.315} C_VEL
LIN {X 0,Y 430.894,Z 535.503,A -85,B 0,C 180,E1 -9790.901,E2 -9790.901} C_VEL
LIN {X 0,Y 430.112,Z 548.627,A -85,B 0,C 180,E1 -9791.656,E2 -9791.656} C_VEL
LIN {X 0,Y 429.217,Z 561.606,A -85,B 0,C 180,E1 -9792.615,E2 -9792.615} C_VEL
LIN {X 0,Y 428.233,Z 573.241,A -85,B 0,C 180,E1 -9793.679,E2 -9793.679} C_VEL
LIN {X 0,Y 427.209,Z 584.88,A -85,B 0,C 180,E1 -9794.985,E2 -9794.985} C_VEL
LIN {X 0,Y 426.365,Z 595.452,A -85,B 0,C 180,E1 -9796.441,E2 -9796.441} C_VEL
LIN {X 0,Y 425.732,Z 603.877,A -85,B 0,C 180,E1 -9797.851,E2 -9797.851} C_VEL
LIN {X 0,Y 425.007,Z 612.098,A -85,B 0,C 180,E1 -9799.521,E2 -9799.521} C_VEL
LIN {X 0,Y 424.656,Z 617.852,A -85,B 0,C 180,E1 -9800.956,E2 -9800.956} C_VEL
LIN {X 0,Y 424.367,Z 622.567,A -85,B 0,C 180,E1 -9802.388,E2 -9802.388} C_VEL
LIN {X 0,Y 424.228,Z 627.458,A -85,B 0,C 180,E1 -9804.297,E2 -9804.297} C_VEL
LIN {X 0,Y 424.072,Z 630.854,A -85,B 0,C 180,E1 -9806.201,E2 -9806.201} C_VEL
LIN {X 0,Y 424.119,Z 632.86,A -85,B 0,C 180,E1 -9808.102,E2 -9808.102} C_VEL
LIN {X 0,Y 424.06,Z 633.522,A -85,B 0,C 180,E1 -9810.001,E2 -9810.001} C_VEL
LIN {X 0,Y 424.119,Z 632.853,A -85,B 0,C 180,E1 -9811.901,E2 -9811.901} C_VEL
LIN {X 0,Y 424.073,Z 630.84,A -85,B 0,C 180,E1 -9813.802,E2 -9813.802} C_VEL
LIN {X 0,Y 424.21,Z 627.44,A -85,B 0,C 180,E1 -9815.706,E2 -9815.706} C_VEL
LIN {X 0,Y 424.333,Z 623.946,A -85,B 0,C 180,E1 -9817.137,E2 -9817.137} C_VEL
LIN {X 0,Y 424.579,Z 619.499,A -85,B 0,C 180,E1 -9818.569,E2 -9818.569} C_VEL
LIN {X 0,Y 424.954,Z 613.078,A -85,B 0,C 180,E1 -9820.242,E2 -9820.242} C_VEL
LIN {X 0,Y 425.633,Z 605.106,A -85,B 0,C 180,E1 -9821.913,E2 -9821.913} C_VEL
LIN {X 0,Y 426.25,Z 596.463,A -85,B 0,C 180,E1 -9823.396,E2 -9823.396} C_VEL
LIN {X 0,Y 427.06,Z 586.72,A -85,B 0,C 180,E1 -9824.78,E2 -9824.78} C_VEL
LIN {X 0,Y 428.052,Z 575.517,A -85,B 0,C 180,E1 -9826.086,E2 -9826.086} C_VEL
LIN {X 0,Y 428.963,Z 564.365,A -85,B 0,C 180,E1 -9827.153,E2 -9827.153} C_VEL
LIN {X 0,Y 429.88,Z 552.222,A -85,B 0,C 180,E1 -9828.098,E2 -9828.098} C_VEL
LIN {X 0,Y 430.724,Z 538.881,A -85,B 0,C 180,E1 -9828.917,E2 -9828.917} C_VEL
LIN {X 0,Y 431.424,Z 524.663,A -85,B 0,C 180,E1 -9829.572,E2 -9829.572} C_VEL
LIN {X 0,Y 432.01,Z 510.871,A -85,B 0,C 180,E1 -9830.009,E2 -9830.009} C_VEL
LIN {X 0,Y 432.435,Z 490.498,A -85,B 0,C 180,E1 -9830.391,E2 -9830.391} C_VEL
LIN {X 0,Y 433.576,Z 396.878,A -85,B 0,C 180,E1 -9831.963,E2 -9831.963} C_VEL
LIN {X 0,Y 428.53,Z 370.69,A -85,B 0,C 180,E1 -9832.715,E2 -9832.715} C_VEL
LIN {X 0,Y 429.27,Z 360.218,A -85,B 0,C 180,E1 -9834.677,E2 -9834.677} C_VEL
LIN {X 0,Y 427.256,Z 349.837,A -85,B 0,C 180,E1 -9836.82,E2 -9836.82} C_VEL
LIN {X 0,Y 425.297,Z 341.133,A -85,B 0,C 180,E1 -9838.701,E2 -9838.701} C_VEL
LIN {X 0,Y 425.269,Z 341.139,A -85,B 0,C 180,E1 -9841.928,E2 -9841.928} C_VEL
LIN {X 0,Y 425.303,Z 341.133,A -85,B 0,C 180,E1 -9845.337,E2 -9845.337} C_VEL
LIN {X 0,Y 425.306,Z 341.13,A -85,B 0,C 180,E1 -9848.899,E2 -9848.899} C_VEL
LIN {X 0,Y 425.295,Z 341.131,A -85,B 0,C 180,E1 -9851.959,E2 -9851.959} C_VEL
LIN {X 0,Y 425.29,Z 341.135,A -85,B 0,C 180,E1 -9855.284,E2 -9855.284} C_VEL
LIN {X 0,Y 425.28,Z 341.135,A -85,B 0,C 180,E1 -9858.622,E2 -9858.622} C_VEL
LIN {X 0,Y 425.314,Z 341.131,A -85,B 0,C 180,E1 -9861.103,E2 -9861.103} C_VEL
LIN {X 0,Y 425.304,Z 341.133,A -85,B 0,C 180,E1 -9864.665,E2 -9864.665} C_VEL
LIN {X 0,Y 425.27,Z 341.139,A -85,B 0,C 180,E1 -9868.074,E2 -9868.074} C_VEL
LIN {X 0,Y 425.319,Z 341.137,A -85,B 0,C 180,E1 -9871.367,E2 -9871.367} C_VEL
LIN {X 0,Y 425.33,Z 341.262,A -85,B 0,C 180,E1 -9873.636,E2 -9873.636} C_VEL
LIN {X 0,Y 428.035,Z 351.673,A -85,B 0,C 180,E1 -9875.765,E2 -9875.765} C_VEL
LIN {X 0,Y 429.225,Z 358.686,A -85,B 0,C 180,E1 -9877.115,E2 -9877.115} C_VEL
LIN {X 0,Y 428.682,Z 375.611,A -85,B 0,C 180,E1 -9880.112,E2 -9880.112} C_VEL
LIN {X 0,Y 428.512,Z 379.586,A -85,B 0,C 180,E1 -9880.82,E2 -9880.82} C_VEL
LIN {X 0,Y 431.742,Z 394.527,A -85,B 0,C 180,E1 -9881.403,E2 -9881.403} C_VEL
LIN {X 0,Y 431.682,Z 404.36,A -85,B 0,C 180,E1 -9881.639,E2 -9881.639} C_VEL
LIN {X 0,Y 429.61,Z 489.82,A -85,B 0,C 180,E1 -9883.517,E2 -9883.517} C_VEL
LIN {X 0,Y 429.153,Z 503.372,A -85,B 0,C 180,E1 -9884.018,E2 -9884.018} C_VEL
LIN {X 0,Y 428.689,Z 515.787,A -85,B 0,C 180,E1 -9884.671,E2 -9884.671} C_VEL
LIN {X 0,Y 428.035,Z 528.051,A -85,B 0,C 180,E1 -9885.524,E2 -9885.524} C_VEL
LIN {X 0,Y 427.435,Z 539.234,A -85,B 0,C 180,E1 -9886.516,E2 -9886.516} C_VEL
LIN {X 0,Y 426.711,Z 549.382,A -85,B 0,C 180,E1 -9887.637,E2 -9887.637} C_VEL
LIN {X 0,Y 426.155,Z 558.14,A -85,B 0,C 180,E1 -9888.827,E2 -9888.827} C_VEL
LIN {X 0,Y 425.597,Z 566.696,A -85,B 0,C 180,E1 -9890.255,E2 -9890.255} C_VEL
LIN {X 0,Y 425.09,Z 573.496,A -85,B 0,C 180,E1 -9891.682,E2 -9891.682} C_VEL
LIN {X 0,Y 424.8,Z 579.7,A -85,B 0,C 180,E1 -9893.35,E2 -9893.35} C_VEL
LIN {X 0,Y 424.424,Z 583.717,A -85,B 0,C 180,E1 -9894.775,E2 -9894.775} C_VEL
LIN {X 0,Y 424.451,Z 586.62,A -85,B 0,C 180,E1 -9896.203,E2 -9896.203} C_VEL
LIN {X 0,Y 424.319,Z 587.985,A -85,B 0,C 180,E1 -9897.152,E2 -9897.152} C_VEL
LIN {X 0,Y 424.22,Z 588.93,A -85,B 0,C 180,E1 -9898.101,E2 -9898.101} C_VEL
LIN {X 0,Y 424.168,Z 589.47,A -85,B 0,C 180,E1 -9899.051,E2 -9899.051} C_VEL
LIN {X 0,Y 424.138,Z 589.555,A -85,B 0,C 180,E1 -9900,E2 -9900} C_VEL
LIN {X 0,Y 424.142,Z 589.212,A -85,B 0,C 180,E1 -9900.95,E2 -9900.95} C_VEL
LIN {X 0,Y 424.197,Z 588.466,A -85,B 0,C 180,E1 -9901.899,E2 -9901.899} C_VEL
LIN {X 0,Y 424.297,Z 587.281,A -85,B 0,C 180,E1 -9902.848,E2 -9902.848} C_VEL
LIN {X 0,Y 424.304,Z 584.675,A -85,B 0,C 180,E1 -9904.275,E2 -9904.275} C_VEL
LIN {X 0,Y 424.474,Z 581.008,A -85,B 0,C 180,E1 -9905.701,E2 -9905.701} C_VEL
LIN {X 0,Y 424.676,Z 575.353,A -85,B 0,C 180,E1 -9907.345,E2 -9907.345} C_VEL
LIN {X 0,Y 424.981,Z 568.922,A -85,B 0,C 180,E1 -9908.799,E2 -9908.799} C_VEL
LIN {X 0,Y 425.417,Z 560.947,A -85,B 0,C 180,E1 -9910.23,E2 -9910.23} C_VEL
LIN {X 0,Y 425.825,Z 552.805,A -85,B 0,C 180,E1 -9911.423,E2 -9911.423} C_VEL
LIN {X 0,Y 426.462,Z 542.909,A -85,B 0,C 180,E1 -9912.613,E2 -9912.613} C_VEL
LIN {X 0,Y 426.937,Z 531.702,A -85,B 0,C 180,E1 -9913.694,E2 -9913.694} C_VEL
LIN {X 0,Y 427.463,Z 521.006,A -85,B 0,C 180,E1 -9914.521,E2 -9914.521} C_VEL
LIN {X 0,Y 427.918,Z 509.277,A -85,B 0,C 180,E1 -9915.235,E2 -9915.235} C_VEL
LIN {X 0,Y 428.344,Z 495.938,A -85,B 0,C 180,E1 -9915.829,E2 -9915.829} C_VEL
LIN {X 0,Y 428.668,Z 483.084,A -85,B 0,C 180,E1 -9916.214,E2 -9916.214} C_VEL
LIN {X 0,Y 429.954,Z 393.781,A -85,B 0,C 180,E1 -9917.985,E2 -9917.985} C_VEL
LIN {X 0,Y 427.086,Z 376.871,A -85,B 0,C 180,E1 -9918.468,E2 -9918.468} C_VEL
LIN {X 0,Y 427.686,Z 358.953,A -85,B 0,C 180,E1 -9921.699,E2 -9921.699} C_VEL
LIN {X 0,Y 427.741,Z 353.961,A -85,B 0,C 180,E1 -9922.608,E2 -9922.608} C_VEL
LIN {X 0,Y 425.662,Z 342.76,A -85,B 0,C 180,E1 -9924.755,E2 -9924.755} C_VEL
LIN {X 0,Y 425.366,Z 341.125,A -85,B 0,C 180,E1 -9925.084,E2 -9925.084} C_VEL
LIN {X 0,Y 425.354,Z 341.126,A -85,B 0,C 180,E1 -9927.557,E2 -9927.557} C_VEL
LIN {X 0,Y 425.294,Z 341.129,A -85,B 0,C 180,E1 -9930.816,E2 -9930.816} C_VEL
LIN {X 0,Y 425.317,Z 341.132,A -85,B 0,C 180,E1 -9934.287,E2 -9934.287} C_VEL
LIN {X 0,Y 425.281,Z 341.137,A -85,B 0,C 180,E1 -9937.694,E2 -9937.694} C_VEL
LIN {X 0,Y 425.252,Z 341.136,A -85,B 0,C 180,E1 -9940.514,E2 -9940.514} C_VEL
LIN {X 0,Y 425.261,Z 341.138,A -85,B 0,C 180,E1 -9943.35,E2 -9943.35} C_VEL
LIN {X 0,Y 425.263,Z 341.138,A -85,B 0,C 180,E1 -9946.043,E2 -9946.043} C_VEL
LIN {X 0,Y 425.256,Z 341.136,A -85,B 0,C 180,E1 -9948.618,E2 -9948.618} C_VEL
LIN {X 0,Y 425.281,Z 341.135,A -85,B 0,C 180,E1 -9951.098,E2 -9951.098} C_VEL
LIN {X 0,Y 425.299,Z 341.131,A -85,B 0,C 180,E1 -9954.663,E2 -9954.663} C_VEL
LIN {X 0,Y 425.252,Z 341.14,A -85,B 0,C 180,E1 -9958.071,E2 -9958.071} C_VEL
LIN {X 0,Y 425.299,Z 341.136,A -85,B 0,C 180,E1 -9961.364,E2 -9961.364} C_VEL
LIN {X 0,Y 425.268,Z 341.205,A -85,B 0,C 180,E1 -9962.579,E2 -9962.579} C_VEL
LIN {X 0,Y 428.16,Z 354.506,A -85,B 0,C 180,E1 -9965.514,E2 -9965.514} C_VEL
LIN {X 0,Y 428.952,Z 359.485,A -85,B 0,C 180,E1 -9966.565,E2 -9966.565} C_VEL
LIN {X 0,Y 428.701,Z 363.732,A -85,B 0,C 180,E1 -9967.365,E2 -9967.365} C_VEL
LIN {X 0,Y 433.769,Z 388.783,A -85,B 0,C 180,E1 -9968.084,E2 -9968.084} C_VEL
LIN {X 0,Y 432.788,Z 463.945,A -85,B 0,C 180,E1 -9969.344,E2 -9969.344} C_VEL
LIN {X 0,Y 432.07,Z 469.797,A -85,B 0,C 180,E1 -9969.407,E2 -9969.407} C_VEL
LIN {X 0,Y 426.347,Z 488.809,A -85,B 0,C 180,E1 -9969.444,E2 -9969.444} C_VEL
LIN {X 0,Y 425.649,Z 494.643,A -85,B 0,C 180,E1 -9969.525,E2 -9969.525} C_VEL
LIN {X 0,Y 425.263,Z 508.16,A -85,B 0,C 180,E1 -9969.849,E2 -9969.849} C_VEL
LIN {X 0,Y 424.635,Z 521.749,A -85,B 0,C 180,E1 -9970.354,E2 -9970.354} C_VEL
LIN {X 0,Y 423.874,Z 535.741,A -85,B 0,C 180,E1 -9971.083,E2 -9971.083} C_VEL
LIN {X 0,Y 422.967,Z 548.788,A -85,B 0,C 180,E1 -9971.971,E2 -9971.971} C_VEL
LIN {X 0,Y 421.966,Z 561.388,A -85,B 0,C 180,E1 -9973.053,E2 -9973.053} C_VEL
LIN {X 0,Y 420.955,Z 572.765,A -85,B 0,C 180,E1 -9974.257,E2 -9974.257} C_VEL
LIN {X 0,Y 420.038,Z 582.192,A -85,B 0,C 180,E1 -9975.463,E2 -9975.463} C_VEL
LIN {X 0,Y 419.317,Z 591.722,A -85,B 0,C 180,E1 -9976.931,E2 -9976.931} C_VEL
LIN {X 0,Y 418.434,Z 600.698,A -85,B 0,C 180,E1 -9978.616,E2 -9978.616} C_VEL
LIN {X 0,Y 417.882,Z 607.976,A -85,B 0,C 180,E1 -9980.317,E2 -9980.317} C_VEL
LIN {X 0,Y 417.531,Z 613.069,A -85,B 0,C 180,E1 -9981.773,E2 -9981.773} C_VEL
LIN {X 0,Y 417.285,Z 618.003,A -85,B 0,C 180,E1 -9983.562,E2 -9983.562} C_VEL
LIN {X 0,Y 417.142,Z 621.292,A -85,B 0,C 180,E1 -9985.166,E2 -9985.166} C_VEL
LIN {X 0,Y 417.032,Z 624.004,A -85,B 0,C 180,E1 -9987.101,E2 -9987.101} C_VEL
LIN {X 0,Y 416.992,Z 625.367,A -85,B 0,C 180,E1 -9989.033,E2 -9989.033} C_VEL
LIN {X 0,Y 416.991,Z 625.405,A -85,B 0,C 180,E1 -9990.964,E2 -9990.964} C_VEL
LIN {X 0,Y 417.031,Z 624.119,A -85,B 0,C 180,E1 -9992.896,E2 -9992.896} C_VEL
LIN {X 0,Y 417.14,Z 621.476,A -85,B 0,C 180,E1 -9994.831,E2 -9994.831} C_VEL
LIN {X 0,Y 417.314,Z 617.404,A -85,B 0,C 180,E1 -9996.769,E2 -9996.769} C_VEL
LIN {X 0,Y 417.637,Z 611.78,A -85,B 0,C 180,E1 -9998.71,E2 -9998.71} C_VEL
LIN {X 0,Y 418.1,Z 605.436,A -85,B 0,C 180,E1 -10000.409,E2 -10000.409} C_VEL
LIN {X 0,Y 418.767,Z 597.544,A -85,B 0,C 180,E1 -10002.108,E2 -10002.108} C_VEL
LIN {X 0,Y 419.497,Z 588.689,A -85,B 0,C 180,E1 -10003.663,E2 -10003.663} C_VEL
LIN {X 0,Y 420.326,Z 579.341,A -85,B 0,C 180,E1 -10005.019,E2 -10005.019} C_VEL
LIN {X 0,Y 421.361,Z 568.268,A -85,B 0,C 180,E1 -10006.346,E2 -10006.346} C_VEL
LIN {X 0,Y 422.298,Z 557.249,A -85,B 0,C 180,E1 -10007.43,E2 -10007.43} C_VEL
LIN {X 0,Y 423.241,Z 545.286,A -85,B 0,C 180,E1 -10008.389,E2 -10008.389} C_VEL
LIN {X 0,Y 424.092,Z 532.076,A -85,B 0,C 180,E1 -10009.227,E2 -10009.227} C_VEL
LIN {X 0,Y 424.824,Z 518.312,A -85,B 0,C 180,E1 -10009.886,E2 -10009.886} C_VEL
LIN {X 0,Y 425.404,Z 504.043,A -85,B 0,C 180,E1 -10010.361,E2 -10010.361} C_VEL
LIN {X 0,Y 425.8,Z 484.144,A -85,B 0,C 180,E1 -10010.752,E2 -10010.752} C_VEL
LIN {X 0,Y 427.175,Z 389.5,A -85,B 0,C 180,E1 -10012.358,E2 -10012.358} C_VEL
LIN {X 0,Y 422.169,Z 365.248,A -85,B 0,C 180,E1 -10013.077,E2 -10013.077} C_VEL
LIN {X 0,Y 421.848,Z 363.462,A -85,B 0,C 180,E1 -10013.156,E2 -10013.156} C_VEL
LIN {X 0,Y 421.857,Z 358.89,A -85,B 0,C 180,E1 -10014.087,E2 -10014.087} C_VEL
LIN {X 0,Y 418.868,Z 344.823,A -85,B 0,C 180,E1 -10017.219,E2 -10017.219} C_VEL
LIN {X 0,Y 418.239,Z 342.015,A -85,B 0,C 180,E1 -10017.88,E2 -10017.88} C_VEL
LIN {X 0,Y 418.232,Z 342.018,A -85,B 0,C 180,E1 -10021.017,E2 -10021.017} C_VEL
LIN {X 0,Y 418.241,Z 342.014,A -85,B 0,C 180,E1 -10023.676,E2 -10023.676} C_VEL
LIN {X 0,Y 418.229,Z 342.015,A -85,B 0,C 180,E1 -10027.223,E2 -10027.223} C_VEL
LIN {X 0,Y 418.198,Z 342.018,A -85,B 0,C 180,E1 -10030.865,E2 -10030.865} C_VEL
LIN {X 0,Y 418.193,Z 342.015,A -85,B 0,C 180,E1 -10033.727,E2 -10033.727} C_VEL
LIN {X 0,Y 418.191,Z 342.018,A -85,B 0,C 180,E1 -10036.446,E2 -10036.446} C_VEL
LIN {X 0,Y 418.197,Z 342.019,A -85,B 0,C 180,E1 -10039.131,E2 -10039.131} C_VEL
LIN {X 0,Y 418.226,Z 342.008,A -85,B 0,C 180,E1 -10042.774,E2 -10042.774} C_VEL
LIN {X 0,Y 418.22,Z 342.011,A -85,B 0,C 180,E1 -10046.32,E2 -10046.32} C_VEL
LIN {X 0,Y 418.227,Z 342.01,A -85,B 0,C 180,E1 -10049.726,E2 -10049.726} C_VEL
LIN {X 0,Y 418.197,Z 342.003,A -85,B 0,C 180,E1 -10053.015,E2 -10053.015} C_VEL
LIN {X 0,Y 418.244,Z 342.008,A -85,B 0,C 180,E1 -10056.216,E2 -10056.216} C_VEL
LIN {X 0,Y 418.235,Z 342.001,A -85,B 0,C 180,E1 -10059.336,E2 -10059.336} C_VEL
LIN {X 0,Y 418.264,Z 341.999,A -85,B 0,C 180,E1 -10062.395,E2 -10062.395} C_VEL
LIN {X 0,Y 418.281,Z 342.003,A -85,B 0,C 180,E1 -10065.402,E2 -10065.402} C_VEL
LIN {X 0,Y 418.297,Z 342.004,A -85,B 0,C 180,E1 -10068.368,E2 -10068.368} C_VEL
LIN {X 0,Y 418.362,Z 341.992,A -85,B 0,C 180,E1 -10071.304,E2 -10071.304} C_VEL
LIN {X 0,Y 418.449,Z 341.986,A -85,B 0,C 180,E1 -10074.216,E2 -10074.216} C_VEL
LIN {X 0,Y 418.522,Z 341.976,A -85,B 0,C 180,E1 -10078.075,E2 -10078.075} C_VEL
LIN {X 0,Y 418.464,Z 341.984,A -85,B 0,C 180,E1 -10080.962,E2 -10080.962} C_VEL
LIN {X 0,Y 418.459,Z 341.983,A -85,B 0,C 180,E1 -10082.888,E2 -10082.888} C_VEL
LIN {X 0,Y 418.471,Z 341.98,A -85,B 0,C 180,E1 -10085.783,E2 -10085.783} C_VEL
LIN {X 0,Y 418.351,Z 341.996,A -85,B 0,C 180,E1 -10088.696,E2 -10088.696} C_VEL
LIN {X 0,Y 418.338,Z 341.998,A -85,B 0,C 180,E1 -10092.615,E2 -10092.615} C_VEL
LIN {X 0,Y 418.286,Z 342.003,A -85,B 0,C 180,E1 -10095.595,E2 -10095.595} C_VEL
LIN {X 0,Y 418.26,Z 342.011,A -85,B 0,C 180,E1 -10098.618,E2 -10098.618} C_VEL
LIN {X 0,Y 418.219,Z 342.003,A -85,B 0,C 180,E1 -10101.697,E2 -10101.697} C_VEL
LIN {X 0,Y 418.23,Z 342.012,A -85,B 0,C 180,E1 -10104.853,E2 -10104.853} C_VEL
LIN {X 0,Y 418.199,Z 342.011,A -85,B 0,C 180,E1 -10108.07,E2 -10108.07} C_VEL
LIN {X 0,Y 418.224,Z 342.012,A -85,B 0,C 180,E1 -10111.02,E2 -10111.02} C_VEL
LIN {X 0,Y 418.219,Z 342.01,A -85,B 0,C 180,E1 -10113.68,E2 -10113.68} C_VEL
LIN {X 0,Y 418.22,Z 342.012,A -85,B 0,C 180,E1 -10117.226,E2 -10117.226} C_VEL
LIN {X 0,Y 418.194,Z 342.015,A -85,B 0,C 180,E1 -10120.868,E2 -10120.868} C_VEL
LIN {X 0,Y 418.189,Z 342.017,A -85,B 0,C 180,E1 -10123.729,E2 -10123.729} C_VEL
LIN {X 0,Y 418.188,Z 342.023,A -85,B 0,C 180,E1 -10126.449,E2 -10126.449} C_VEL
LIN {X 0,Y 418.195,Z 342.017,A -85,B 0,C 180,E1 -10129.135,E2 -10129.135} C_VEL
LIN {X 0,Y 418.223,Z 342.016,A -85,B 0,C 180,E1 -10132.776,E2 -10132.776} C_VEL
LIN {X 0,Y 418.224,Z 342.018,A -85,B 0,C 180,E1 -10136.323,E2 -10136.323} C_VEL
LIN {X 0,Y 418.232,Z 342.014,A -85,B 0,C 180,E1 -10139.729,E2 -10139.729} C_VEL
LIN {X 0,Y 418.272,Z 342.134,A -85,B 0,C 180,E1 -10140.997,E2 -10140.997} C_VEL
LIN {X 0,Y 420.775,Z 353.482,A -85,B 0,C 180,E1 -10143.464,E2 -10143.464} C_VEL
LIN {X 0,Y 422.423,Z 361.548,A -85,B 0,C 180,E1 -10145.161,E2 -10145.161} C_VEL
LIN {X 0,Y 421.767,Z 370.812,A -85,B 0,C 180,E1 -10146.912,E2 -10146.912} C_VEL
LIN {X 0,Y 427.046,Z 397.937,A -85,B 0,C 180,E1 -10147.697,E2 -10147.697} C_VEL
LIN {X 0,Y 425.471,Z 507.626,A -85,B 0,C 180,E1 -10149.579,E2 -10149.579} C_VEL
LIN {X 0,Y 424.916,Z 521.746,A -85,B 0,C 180,E1 -10149.993,E2 -10149.993} C_VEL
LIN {X 0,Y 424.187,Z 535.441,A -85,B 0,C 180,E1 -10150.587,E2 -10150.587} C_VEL
LIN {X 0,Y 423.341,Z 548.996,A -85,B 0,C 180,E1 -10151.383,E2 -10151.383} C_VEL
LIN {X 0,Y 422.432,Z 561.543,A -85,B 0,C 180,E1 -10152.326,E2 -10152.326} C_VEL
LIN {X 0,Y 421.413,Z 573.177,A -85,B 0,C 180,E1 -10153.407,E2 -10153.407} C_VEL
LIN {X 0,Y 420.536,Z 582.862,A -85,B 0,C 180,E1 -10154.493,E2 -10154.493} C_VEL
LIN {X 0,Y 419.541,Z 593.594,A -85,B 0,C 180,E1 -10155.944,E2 -10155.944} C_VEL
LIN {X 0,Y 418.833,Z 602.455,A -85,B 0,C 180,E1 -10157.402,E2 -10157.402} C_VEL
LIN {X 0,Y 418.11,Z 610.946,A -85,B 0,C 180,E1 -10159.101,E2 -10159.101} C_VEL
LIN {X 0,Y 417.598,Z 617.786,A -85,B 0,C 180,E1 -10160.802,E2 -10160.802} C_VEL
LIN {X 0,Y 417.315,Z 622.5,A -85,B 0,C 180,E1 -10162.259,E2 -10162.259} C_VEL
LIN {X 0,Y 417.141,Z 627.391,A -85,B 0,C 180,E1 -10164.2,E2 -10164.2} C_VEL
LIN {X 0,Y 416.989,Z 630.787,A -85,B 0,C 180,E1 -10166.136,E2 -10166.136} C_VEL
LIN {X 0,Y 417.027,Z 632.793,A -85,B 0,C 180,E1 -10168.07,E2 -10168.07} C_VEL
LIN {X 0,Y 416.981,Z 633.455,A -85,B 0,C 180,E1 -10170.001,E2 -10170.001} C_VEL
LIN {X 0,Y 417.027,Z 632.786,A -85,B 0,C 180,E1 -10171.933,E2 -10171.933} C_VEL
LIN {X 0,Y 416.99,Z 630.772,A -85,B 0,C 180,E1 -10173.867,E2 -10173.867} C_VEL
LIN {X 0,Y 417.13,Z 627.372,A -85,B 0,C 180,E1 -10175.803,E2 -10175.803} C_VEL
LIN {X 0,Y 417.318,Z 622.48,A -85,B 0,C 180,E1 -10177.744,E2 -10177.744} C_VEL
LIN {X 0,Y 417.735,Z 615.946,A -85,B 0,C 180,E1 -10179.687,E2 -10179.687} C_VEL
LIN {X 0,Y 418.323,Z 608.675,A -85,B 0,C 180,E1 -10181.387,E2 -10181.387} C_VEL
LIN {X 0,Y 418.984,Z 600.209,A -85,B 0,C 180,E1 -10182.996,E2 -10182.996} C_VEL
LIN {X 0,Y 419.831,Z 590.218,A -85,B 0,C 180,E1 -10184.544,E2 -10184.544} C_VEL
LIN {X 0,Y 420.789,Z 579.756,A -85,B 0,C 180,E1 -10185.874,E2 -10185.874} C_VEL
LIN {X 0,Y 421.825,Z 568.207,A -85,B 0,C 180,E1 -10187.078,E2 -10187.078} C_VEL
LIN {X 0,Y 422.853,Z 555.392,A -85,B 0,C 180,E1 -10188.159,E2 -10188.159} C_VEL
LIN {X 0,Y 423.73,Z 543.313,A -85,B 0,C 180,E1 -10188.97,E2 -10188.97} C_VEL
LIN {X 0,Y 424.45,Z 530.255,A -85,B 0,C 180,E1 -10189.655,E2 -10189.655} C_VEL
LIN {X 0,Y 425.188,Z 516.114,A -85,B 0,C 180,E1 -10190.186,E2 -10190.186} C_VEL
LIN {X 0,Y 425.556,Z 502.694,A -85,B 0,C 180,E1 -10190.515,E2 -10190.515} C_VEL
LIN {X 0,Y 427.033,Z 399.331,A -85,B 0,C 180,E1 -10192.272,E2 -10192.272} C_VEL
LIN {X 0,Y 425.906,Z 391.669,A -85,B 0,C 180,E1 -10192.471,E2 -10192.471} C_VEL
LIN {X 0,Y 421.73,Z 370.59,A -85,B 0,C 180,E1 -10193.109,E2 -10193.109} C_VEL
LIN {X 0,Y 422.355,Z 361.489,A -85,B 0,C 180,E1 -10194.846,E2 -10194.846} C_VEL
LIN {X 0,Y 420.058,Z 349.911,A -85,B 0,C 180,E1 -10197.289,E2 -10197.289} C_VEL
LIN {X 0,Y 418.26,Z 342.01,A -85,B 0,C 180,E1 -10199.047,E2 -10199.047} C_VEL
LIN {X 0,Y 418.25,Z 342.011,A -85,B 0,C 180,E1 -10202.529,E2 -10202.529} C_VEL
LIN {X 0,Y 418.263,Z 342.008,A -85,B 0,C 180,E1 -10204.842,E2 -10204.842} C_VEL
LIN {X 0,Y 418.255,Z 342.007,A -85,B 0,C 180,E1 -10208.443,E2 -10208.443} C_VEL
LIN {X 0,Y 418.227,Z 342.013,A -85,B 0,C 180,E1 -10210.949,E2 -10210.949} C_VEL
LIN {X 0,Y 418.215,Z 342.014,A -85,B 0,C 180,E1 -10213.73,E2 -10213.73} C_VEL
LIN {X 0,Y 418.214,Z 342.014,A -85,B 0,C 180,E1 -10216.449,E2 -10216.449} C_VEL
LIN {X 0,Y 418.228,Z 342.014,A -85,B 0,C 180,E1 -10219.131,E2 -10219.131} C_VEL
LIN {X 0,Y 418.233,Z 342.012,A -85,B 0,C 180,E1 -10222.167,E2 -10222.167} C_VEL
LIN {X 0,Y 418.27,Z 342.007,A -85,B 0,C 180,E1 -10225.42,E2 -10225.42} C_VEL
LIN {X 0,Y 418.217,Z 342.02,A -85,B 0,C 180,E1 -10228.604,E2 -10228.604} C_VEL
LIN {X 0,Y 418.252,Z 342.018,A -85,B 0,C 180,E1 -10231.934,E2 -10231.934} C_VEL
LIN {X 0,Y 418.25,Z 342.085,A -85,B 0,C 180,E1 -10233.087,E2 -10233.087} C_VEL
LIN {X 0,Y 421.165,Z 352.818,A -85,B 0,C 180,E1 -10235.344,E2 -10235.344} C_VEL
LIN {X 0,Y 422.488,Z 359.747,A -85,B 0,C 180,E1 -10236.729,E2 -10236.729} C_VEL
LIN {X 0,Y 422.254,Z 371.006,A -85,B 0,C 180,E1 -10238.761,E2 -10238.761} C_VEL
LIN {X 0,Y 421.885,Z 380.071,A -85,B 0,C 180,E1 -10240.381,E2 -10240.381} C_VEL
LIN {X 0,Y 425.226,Z 395.109,A -85,B 0,C 180,E1 -10241.002,E2 -10241.002} C_VEL
LIN {X 0,Y 425.386,Z 399.313,A -85,B 0,C 180,E1 -10241.121,E2 -10241.121} C_VEL
LIN {X 0,Y 422.958,Z 490.107,A -85,B 0,C 180,E1 -10243.188,E2 -10243.188} C_VEL
LIN {X 0,Y 422.473,Z 503.616,A -85,B 0,C 180,E1 -10243.697,E2 -10243.697} C_VEL
LIN {X 0,Y 421.941,Z 517.009,A -85,B 0,C 180,E1 -10244.42,E2 -10244.42} C_VEL
LIN {X 0,Y 421.233,Z 529.038,A -85,B 0,C 180,E1 -10245.285,E2 -10245.285} C_VEL
LIN {X 0,Y 420.588,Z 540.135,A -85,B 0,C 180,E1 -10246.297,E2 -10246.297} C_VEL
LIN {X 0,Y 419.817,Z 550.123,A -85,B 0,C 180,E1 -10247.43,E2 -10247.43} C_VEL
LIN {X 0,Y 419.225,Z 558.822,A -85,B 0,C 180,E1 -10248.64,E2 -10248.64} C_VEL
LIN {X 0,Y 418.636,Z 567.302,A -85,B 0,C 180,E1 -10250.092,E2 -10250.092} C_VEL
LIN {X 0,Y 418.149,Z 573.055,A -85,B 0,C 180,E1 -10251.3,E2 -10251.3} C_VEL
LIN {X 0,Y 417.774,Z 579.438,A -85,B 0,C 180,E1 -10252.997,E2 -10252.997} C_VEL
LIN {X 0,Y 417.373,Z 584.195,A -85,B 0,C 180,E1 -10254.686,E2 -10254.686} C_VEL
LIN {X 0,Y 417.393,Z 587.057,A -85,B 0,C 180,E1 -10256.138,E2 -10256.138} C_VEL
LIN {X 0,Y 417.257,Z 588.393,A -85,B 0,C 180,E1 -10257.104,E2 -10257.104} C_VEL
LIN {X 0,Y 417.146,Z 589.32,A -85,B 0,C 180,E1 -10258.069,E2 -10258.069} C_VEL
LIN {X 0,Y 417.087,Z 589.836,A -85,B 0,C 180,E1 -10259.035,E2 -10259.035} C_VEL
LIN {X 0,Y 417.055,Z 589.883,A -85,B 0,C 180,E1 -10260,E2 -10260} C_VEL
LIN {X 0,Y 417.062,Z 589.515,A -85,B 0,C 180,E1 -10260.966,E2 -10260.966} C_VEL
LIN {X 0,Y 417.124,Z 588.742,A -85,B 0,C 180,E1 -10261.931,E2 -10261.931} C_VEL
LIN {X 0,Y 417.23,Z 587.509,A -85,B 0,C 180,E1 -10262.897,E2 -10262.897} C_VEL
LIN {X 0,Y 417.219,Z 584.847,A -85,B 0,C 180,E1 -10264.347,E2 -10264.347} C_VEL
LIN {X 0,Y 417.412,Z 581.117,A -85,B 0,C 180,E1 -10265.798,E2 -10265.798} C_VEL
LIN {X 0,Y 417.587,Z 576.221,A -85,B 0,C 180,E1 -10267.252,E2 -10267.252} C_VEL
LIN {X 0,Y 417.889,Z 570.018,A -85,B 0,C 180,E1 -10268.706,E2 -10268.706} C_VEL
LIN {X 0,Y 418.322,Z 562.267,A -85,B 0,C 180,E1 -10270.161,E2 -10270.161} C_VEL
LIN {X 0,Y 418.842,Z 552.524,A -85,B 0,C 180,E1 -10271.616,E2 -10271.616} C_VEL
LIN {X 0,Y 419.508,Z 542.452,A -85,B 0,C 180,E1 -10272.825,E2 -10272.825} C_VEL
LIN {X 0,Y 420.024,Z 530.741,A -85,B 0,C 180,E1 -10273.954,E2 -10273.954} C_VEL
LIN {X 0,Y 420.523,Z 520.159,A -85,B 0,C 180,E1 -10274.766,E2 -10274.766} C_VEL
LIN {X 0,Y 421.025,Z 507.992,A -85,B 0,C 180,E1 -10275.491,E2 -10275.491} C_VEL
LIN {X 0,Y 421.524,Z 494.167,A -85,B 0,C 180,E1 -10276.092,E2 -10276.092} C_VEL
LIN {X 0,Y 421.763,Z 479.754,A -85,B 0,C 180,E1 -10276.487,E2 -10276.487} C_VEL
LIN {X 0,Y 423.102,Z 394.845,A -85,B 0,C 180,E1 -10278.208,E2 -10278.208} C_VEL
LIN {X 0,Y 420.143,Z 377.104,A -85,B 0,C 180,E1 -10278.721,E2 -10278.721} C_VEL
LIN {X 0,Y 420.852,Z 357.263,A -85,B 0,C 180,E1 -10282.328,E2 -10282.328} C_VEL
LIN {X 0,Y 420.266,Z 351.927,A -85,B 0,C 180,E1 -10283.341,E2 -10283.341} C_VEL
LIN {X 0,Y 418.316,Z 342.003,A -85,B 0,C 180,E1 -10285.294,E2 -10285.294} C_VEL
LIN {X 0,Y 418.297,Z 342.008,A -85,B 0,C 180,E1 -10288.063,E2 -10288.063} C_VEL
LIN {X 0,Y 418.217,Z 342.011,A -85,B 0,C 180,E1 -10291.396,E2 -10291.396} C_VEL
LIN {X 0,Y 418.271,Z 342.007,A -85,B 0,C 180,E1 -10294.58,E2 -10294.58} C_VEL
LIN {X 0,Y 418.227,Z 342.017,A -85,B 0,C 180,E1 -10297.832,E2 -10297.832} C_VEL
LIN {X 0,Y 418.215,Z 342.012,A -85,B 0,C 180,E1 -10300.949,E2 -10300.949} C_VEL
LIN {X 0,Y 418.215,Z 342.018,A -85,B 0,C 180,E1 -10303.729,E2 -10303.729} C_VEL
LIN {X 0,Y 418.207,Z 342.015,A -85,B 0,C 180,E1 -10306.447,E2 -10306.447} C_VEL
LIN {X 0,Y 418.213,Z 342.015,A -85,B 0,C 180,E1 -10309.132,E2 -10309.132} C_VEL
LIN {X 0,Y 418.239,Z 342.012,A -85,B 0,C 180,E1 -10312.774,E2 -10312.774} C_VEL
LIN {X 0,Y 418.234,Z 342.013,A -85,B 0,C 180,E1 -10316.32,E2 -10316.32} C_VEL
LIN {X 0,Y 418.242,Z 342.013,A -85,B 0,C 180,E1 -10319.726,E2 -10319.726} C_VEL
LIN {X 0,Y 418.236,Z 342.077,A -85,B 0,C 180,E1 -10322.249,E2 -10322.249} C_VEL
LIN {X 0,Y 420.82,Z 353.956,A -85,B 0,C 180,E1 -10324.93,E2 -10324.93} C_VEL
LIN {X 0,Y 422.06,Z 360.949,A -85,B 0,C 180,E1 -10326.443,E2 -10326.443} C_VEL
LIN {X 0,Y 421.866,Z 363.595,A -85,B 0,C 180,E1 -10326.969,E2 -10326.969} C_VEL
LIN {X 0,Y 427.127,Z 388.964,A -85,B 0,C 180,E1 -10327.726,E2 -10327.726} C_VEL
LIN {X 0,Y 425.649,Z 494.643,A -85,B 0,C 180,E1 -10329.525,E2 -10329.525} C_VEL
LIN {X 0,Y 425.265,Z 498.534,A -85,B 0,C 180,E1 -10329.587,E2 -10329.587} C_VEL
LIN {X 0,Y 423.194,Z 506.143,A -85,B 0,C 180,E1 -10329.682,E2 -10329.682} C_VEL
LIN {X 0,Y 418.7,Z 519.182,A -85,B 0,C 180,E1 -10329.942,E2 -10329.942} C_VEL
LIN {X 0,Y 417.82,Z 524.744,A -85,B 0,C 180,E1 -10330.164,E2 -10330.164} C_VEL
LIN {X 0,Y 416.991,Z 538.378,A -85,B 0,C 180,E1 -10330.924,E2 -10330.924} C_VEL
LIN {X 0,Y 416.098,Z 550.44,A -85,B 0,C 180,E1 -10331.791,E2 -10331.791} C_VEL
LIN {X 0,Y 415.055,Z 562.737,A -85,B 0,C 180,E1 -10332.889,E2 -10332.889} C_VEL
LIN {X 0,Y 414.112,Z 572.836,A -85,B 0,C 180,E1 -10333.99,E2 -10333.99} C_VEL
LIN {X 0,Y 413.144,Z 582.263,A -85,B 0,C 180,E1 -10335.215,E2 -10335.215} C_VEL
LIN {X 0,Y 412.347,Z 592.077,A -85,B 0,C 180,E1 -10336.755,E2 -10336.755} C_VEL
LIN {X 0,Y 411.466,Z 600.768,A -85,B 0,C 180,E1 -10338.421,E2 -10338.421} C_VEL
LIN {X 0,Y 410.854,Z 608.045,A -85,B 0,C 180,E1 -10340.149,E2 -10340.149} C_VEL
LIN {X 0,Y 410.373,Z 614.581,A -85,B 0,C 180,E1 -10342.124,E2 -10342.124} C_VEL
LIN {X 0,Y 410.124,Z 619.477,A -85,B 0,C 180,E1 -10344.097,E2 -10344.097} C_VEL
LIN {X 0,Y 409.943,Z 622.889,A -85,B 0,C 180,E1 -10346.066,E2 -10346.066} C_VEL
LIN {X 0,Y 409.967,Z 624.919,A -85,B 0,C 180,E1 -10348.034,E2 -10348.034} C_VEL
LIN {X 0,Y 409.905,Z 625.618,A -85,B 0,C 180,E1 -10349.999,E2 -10349.999} C_VEL
LIN {X 0,Y 409.965,Z 624.995,A -85,B 0,C 180,E1 -10351.963,E2 -10351.963} C_VEL
LIN {X 0,Y 409.941,Z 623.037,A -85,B 0,C 180,E1 -10353.931,E2 -10353.931} C_VEL
LIN {X 0,Y 410.073,Z 621.542,A -85,B 0,C 180,E1 -10354.914,E2 -10354.914} C_VEL
LIN {X 0,Y 410.25,Z 617.47,A -85,B 0,C 180,E1 -10356.886,E2 -10356.886} C_VEL
LIN {X 0,Y 410.579,Z 611.846,A -85,B 0,C 180,E1 -10358.86,E2 -10358.86} C_VEL
LIN {X 0,Y 411.05,Z 605.502,A -85,B 0,C 180,E1 -10360.59,E2 -10360.59} C_VEL
LIN {X 0,Y 411.801,Z 597.609,A -85,B 0,C 180,E1 -10362.316,E2 -10362.316} C_VEL
LIN {X 0,Y 412.501,Z 589.353,A -85,B 0,C 180,E1 -10363.798,E2 -10363.798} C_VEL
LIN {X 0,Y 413.441,Z 579.406,A -85,B 0,C 180,E1 -10365.275,E2 -10365.275} C_VEL
LIN {X 0,Y 414.533,Z 568.332,A -85,B 0,C 180,E1 -10366.623,E2 -10366.623} C_VEL
LIN {X 0,Y 415.515,Z 557.311,A -85,B 0,C 180,E1 -10367.723,E2 -10367.723} C_VEL
LIN {X 0,Y 416.507,Z 545.347,A -85,B 0,C 180,E1 -10368.697,E2 -10368.697} C_VEL
LIN {X 0,Y 417.357,Z 532.673,A -85,B 0,C 180,E1 -10369.52,E2 -10369.52} C_VEL
LIN {X 0,Y 418.172,Z 518.368,A -85,B 0,C 180,E1 -10370.216,E2 -10370.216} C_VEL
LIN {X 0,Y 418.771,Z 504.093,A -85,B 0,C 180,E1 -10370.698,E2 -10370.698} C_VEL
LIN {X 0,Y 419.19,Z 484.185,A -85,B 0,C 180,E1 -10371.095,E2 -10371.095} C_VEL
LIN {X 0,Y 420.616,Z 391.146,A -85,B 0,C 180,E1 -10372.697,E2 -10372.697} C_VEL
LIN {X 0,Y 416.475,Z 369.971,A -85,B 0,C 180,E1 -10373.325,E2 -10373.325} C_VEL
LIN {X 0,Y 415.064,Z 363.654,A -85,B 0,C 180,E1 -10373.531,E2 -10373.531} C_VEL
LIN {X 0,Y 414.931,Z 360.233,A -85,B 0,C 180,E1 -10374.249,E2 -10374.249} C_VEL
LIN {X 0,Y 412.085,Z 346.889,A -85,B 0,C 180,E1 -10377.272,E2 -10377.272} C_VEL
LIN {X 0,Y 411.206,Z 342.891,A -85,B 0,C 180,E1 -10378.241,E2 -10378.241} C_VEL
LIN {X 0,Y 411.175,Z 342.898,A -85,B 0,C 180,E1 -10381.281,E2 -10381.281} C_VEL
LIN {X 0,Y 411.198,Z 342.892,A -85,B 0,C 180,E1 -10384.332,E2 -10384.332} C_VEL
LIN {X 0,Y 411.177,Z 342.89,A -85,B 0,C 180,E1 -10387.973,E2 -10387.973} C_VEL
LIN {X 0,Y 411.138,Z 342.898,A -85,B 0,C 180,E1 -10391.224,E2 -10391.224} C_VEL
LIN {X 0,Y 411.164,Z 342.893,A -85,B 0,C 180,E1 -10394.489,E2 -10394.489} C_VEL
LIN {X 0,Y 411.151,Z 342.893,A -85,B 0,C 180,E1 -10398.191,E2 -10398.191} C_VEL
LIN {X 0,Y 411.183,Z 342.88,A -85,B 0,C 180,E1 -10401.832,E2 -10401.832} C_VEL
LIN {X 0,Y 411.191,Z 342.889,A -85,B 0,C 180,E1 -10405.122,E2 -10405.122} C_VEL
LIN {X 0,Y 411.15,Z 342.883,A -85,B 0,C 180,E1 -10408.001,E2 -10408.001} C_VEL
LIN {X 0,Y 411.162,Z 342.889,A -85,B 0,C 180,E1 -10411.406,E2 -10411.406} C_VEL
LIN {X 0,Y 411.174,Z 342.886,A -85,B 0,C 180,E1 -10414.94,E2 -10414.94} C_VEL
LIN {X 0,Y 411.19,Z 342.887,A -85,B 0,C 180,E1 -10417.912,E2 -10417.912} C_VEL
LIN {X 0,Y 411.204,Z 342.873,A -85,B 0,C 180,E1 -10421.05,E2 -10421.05} C_VEL
LIN {X 0,Y 411.235,Z 342.882,A -85,B 0,C 180,E1 -10424.131,E2 -10424.131} C_VEL
LIN {X 0,Y 411.288,Z 342.875,A -85,B 0,C 180,E1 -10427.165,E2 -10427.165} C_VEL
LIN {X 0,Y 411.273,Z 342.878,A -85,B 0,C 180,E1 -10430.161,E2 -10430.161} C_VEL
LIN {X 0,Y 411.37,Z 342.866,A -85,B 0,C 180,E1 -10433.131,E2 -10433.131} C_VEL
LIN {X 0,Y 411.272,Z 342.874,A -85,B 0,C 180,E1 -10435.098,E2 -10435.098} C_VEL
LIN {X 0,Y 411.49,Z 342.852,A -85,B 0,C 180,E1 -10438.042,E2 -10438.042} C_VEL
LIN {X 0,Y 411.487,Z 342.851,A -85,B 0,C 180,E1 -10441.957,E2 -10441.957} C_VEL
LIN {X 0,Y 411.416,Z 342.859,A -85,B 0,C 180,E1 -10445.883,E2 -10445.883} C_VEL
LIN {X 0,Y 411.291,Z 342.876,A -85,B 0,C 180,E1 -10448.847,E2 -10448.847} C_VEL
LIN {X 0,Y 411.258,Z 342.879,A -85,B 0,C 180,E1 -10451.833,E2 -10451.833} C_VEL
LIN {X 0,Y 411.244,Z 342.883,A -85,B 0,C 180,E1 -10454.853,E2 -10454.853} C_VEL
LIN {X 0,Y 411.23,Z 342.882,A -85,B 0,C 180,E1 -10457.916,E2 -10457.916} C_VEL
LIN {X 0,Y 411.182,Z 342.88,A -85,B 0,C 180,E1 -10461.035,E2 -10461.035} C_VEL
LIN {X 0,Y 411.176,Z 342.886,A -85,B 0,C 180,E1 -10464.219,E2 -10464.219} C_VEL
LIN {X 0,Y 411.135,Z 342.891,A -85,B 0,C 180,E1 -10467.487,E2 -10467.487} C_VEL
LIN {X 0,Y 411.182,Z 342.879,A -85,B 0,C 180,E1 -10469.714,E2 -10469.714} C_VEL
LIN {X 0,Y 411.191,Z 342.885,A -85,B 0,C 180,E1 -10473.157,E2 -10473.157} C_VEL
LIN {X 0,Y 411.176,Z 342.894,A -85,B 0,C 180,E1 -10476.553,E2 -10476.553} C_VEL
LIN {X 0,Y 411.155,Z 342.894,A -85,B 0,C 180,E1 -10479.721,E2 -10479.721} C_VEL
LIN {X 0,Y 411.149,Z 342.893,A -85,B 0,C 180,E1 -10483.137,E2 -10483.137} C_VEL
LIN {X 0,Y 411.152,Z 342.896,A -85,B 0,C 180,E1 -10485.883,E2 -10485.883} C_VEL
LIN {X 0,Y 411.146,Z 342.896,A -85,B 0,C 180,E1 -10489.494,E2 -10489.494} C_VEL
LIN {X 0,Y 411.168,Z 342.897,A -85,B 0,C 180,E1 -10492.026,E2 -10492.026} C_VEL
LIN {X 0,Y 411.193,Z 342.89,A -85,B 0,C 180,E1 -10495.125,E2 -10495.125} C_VEL
LIN {X 0,Y 411.155,Z 342.896,A -85,B 0,C 180,E1 -10498.004,E2 -10498.004} C_VEL
LIN {X 0,Y 411.224,Z 343.007,A -85,B 0,C 180,E1 -10500.647,E2 -10500.647} C_VEL
LIN {X 0,Y 414.123,Z 356.103,A -85,B 0,C 180,E1 -10503.548,E2 -10503.548} C_VEL
LIN {X 0,Y 415.487,Z 362.82,A -85,B 0,C 180,E1 -10504.986,E2 -10504.986} C_VEL
LIN {X 0,Y 414.946,Z 370.635,A -85,B 0,C 180,E1 -10506.505,E2 -10506.505} C_VEL
LIN {X 0,Y 420.388,Z 398.426,A -85,B 0,C 180,E1 -10507.334,E2 -10507.334} C_VEL
LIN {X 0,Y 419.305,Z 481.937,A -85,B 0,C 180,E1 -10508.783,E2 -10508.783} C_VEL
LIN {X 0,Y 418.783,Z 508.781,A -85,B 0,C 180,E1 -10509.27,E2 -10509.27} C_VEL
LIN {X 0,Y 418.17,Z 523.211,A -85,B 0,C 180,E1 -10509.72,E2 -10509.72} C_VEL
LIN {X 0,Y 417.423,Z 536.51,A -85,B 0,C 180,E1 -10510.324,E2 -10510.324} C_VEL
LIN {X 0,Y 416.576,Z 549.369,A -85,B 0,C 180,E1 -10511.1,E2 -10511.1} C_VEL
LIN {X 0,Y 415.653,Z 561.479,A -85,B 0,C 180,E1 -10512.028,E2 -10512.028} C_VEL
LIN {X 0,Y 414.583,Z 573.112,A -85,B 0,C 180,E1 -10513.126,E2 -10513.126} C_VEL
LIN {X 0,Y 413.673,Z 582.797,A -85,B 0,C 180,E1 -10514.229,E2 -10514.229} C_VEL
LIN {X 0,Y 412.602,Z 593.528,A -85,B 0,C 180,E1 -10515.703,E2 -10515.703} C_VEL
LIN {X 0,Y 411.856,Z 602.389,A -85,B 0,C 180,E1 -10517.185,E2 -10517.185} C_VEL
LIN {X 0,Y 411.084,Z 610.88,A -85,B 0,C 180,E1 -10518.913,E2 -10518.913} C_VEL
LIN {X 0,Y 410.558,Z 617.719,A -85,B 0,C 180,E1 -10520.642,E2 -10520.642} C_VEL
LIN {X 0,Y 410.256,Z 622.434,A -85,B 0,C 180,E1 -10522.125,E2 -10522.125} C_VEL
LIN {X 0,Y 410.057,Z 627.324,A -85,B 0,C 180,E1 -10524.099,E2 -10524.099} C_VEL
LIN {X 0,Y 409.909,Z 630.72,A -85,B 0,C 180,E1 -10526.069,E2 -10526.069} C_VEL
LIN {X 0,Y 409.923,Z 632.726,A -85,B 0,C 180,E1 -10528.036,E2 -10528.036} C_VEL
LIN {X 0,Y 409.904,Z 633.388,A -85,B 0,C 180,E1 -10530.001,E2 -10530.001} C_VEL
LIN {X 0,Y 409.923,Z 632.718,A -85,B 0,C 180,E1 -10531.966,E2 -10531.966} C_VEL
LIN {X 0,Y 409.909,Z 630.705,A -85,B 0,C 180,E1 -10533.934,E2 -10533.934} C_VEL
LIN {X 0,Y 410.053,Z 627.304,A -85,B 0,C 180,E1 -10535.904,E2 -10535.904} C_VEL
LIN {X 0,Y 410.259,Z 622.412,A -85,B 0,C 180,E1 -10537.878,E2 -10537.878} C_VEL
LIN {X 0,Y 410.706,Z 615.877,A -85,B 0,C 180,E1 -10539.854,E2 -10539.854} C_VEL
LIN {X 0,Y 411.336,Z 608.606,A -85,B 0,C 180,E1 -10541.583,E2 -10541.583} C_VEL
LIN {X 0,Y 411.969,Z 600.702,A -85,B 0,C 180,E1 -10543.118,E2 -10543.118} C_VEL
LIN {X 0,Y 412.773,Z 591.841,A -85,B 0,C 180,E1 -10544.546,E2 -10544.546} C_VEL
LIN {X 0,Y 413.826,Z 580.753,A -85,B 0,C 180,E1 -10546.021,E2 -10546.021} C_VEL
LIN {X 0,Y 414.903,Z 569.429,A -85,B 0,C 180,E1 -10547.245,E2 -10547.245} C_VEL
LIN {X 0,Y 415.958,Z 556.903,A -85,B 0,C 180,E1 -10548.343,E2 -10548.343} C_VEL
LIN {X 0,Y 416.92,Z 544.602,A -85,B 0,C 180,E1 -10549.204,E2 -10549.204} C_VEL
LIN {X 0,Y 417.683,Z 531.482,A -85,B 0,C 180,E1 -10549.923,E2 -10549.923} C_VEL
LIN {X 0,Y 418.506,Z 516.953,A -85,B 0,C 180,E1 -10550.49,E2 -10550.49} C_VEL
LIN {X 0,Y 418.854,Z 504.116,A -85,B 0,C 180,E1 -10550.826,E2 -10550.826} C_VEL
LIN {X 0,Y 420.429,Z 404.458,A -85,B 0,C 180,E1 -10552.547,E2 -10552.547} C_VEL
LIN {X 0,Y 420.226,Z 397.648,A -85,B 0,C 180,E1 -10552.682,E2 -10552.682} C_VEL
LIN {X 0,Y 414.916,Z 370.52,A -85,B 0,C 180,E1 -10553.51,E2 -10553.51} C_VEL
LIN {X 0,Y 415.466,Z 362.76,A -85,B 0,C 180,E1 -10555.019,E2 -10555.019} C_VEL
LIN {X 0,Y 412.883,Z 350.191,A -85,B 0,C 180,E1 -10557.732,E2 -10557.732} C_VEL
LIN {X 0,Y 411.204,Z 342.891,A -85,B 0,C 180,E1 -10559.421,E2 -10559.421} C_VEL
LIN {X 0,Y 411.211,Z 342.887,A -85,B 0,C 180,E1 -10563.157,E2 -10563.157} C_VEL
LIN {X 0,Y 411.197,Z 342.887,A -85,B 0,C 180,E1 -10566.553,E2 -10566.553} C_VEL
LIN {X 0,Y 411.216,Z 342.885,A -85,B 0,C 180,E1 -10569.728,E2 -10569.728} C_VEL
LIN {X 0,Y 411.178,Z 342.894,A -85,B 0,C 180,E1 -10573.134,E2 -10573.134} C_VEL
LIN {X 0,Y 411.173,Z 342.892,A -85,B 0,C 180,E1 -10575.882,E2 -10575.882} C_VEL
LIN {X 0,Y 411.169,Z 342.893,A -85,B 0,C 180,E1 -10578.772,E2 -10578.772} C_VEL
LIN {X 0,Y 411.21,Z 342.886,A -85,B 0,C 180,E1 -10581.832,E2 -10581.832} C_VEL
LIN {X 0,Y 411.216,Z 342.886,A -85,B 0,C 180,E1 -10585.122,E2 -10585.122} C_VEL
LIN {X 0,Y 411.171,Z 342.895,A -85,B 0,C 180,E1 -10588.003,E2 -10588.003} C_VEL
LIN {X 0,Y 411.199,Z 342.896,A -85,B 0,C 180,E1 -10591.409,E2 -10591.409} C_VEL
LIN {X 0,Y 411.221,Z 343.062,A -85,B 0,C 180,E1 -10592.52,E2 -10592.52} C_VEL
LIN {X 0,Y 414.327,Z 354.033,A -85,B 0,C 180,E1 -10594.909,E2 -10594.909} C_VEL
LIN {X 0,Y 415.704,Z 360.682,A -85,B 0,C 180,E1 -10596.289,E2 -10596.289} C_VEL
LIN {X 0,Y 415.931,Z 365.181,A -85,B 0,C 180,E1 -10597.131,E2 -10597.131} C_VEL
LIN {X 0,Y 415.301,Z 380.37,A -85,B 0,C 180,E1 -10599.895,E2 -10599.895} C_VEL
LIN {X 0,Y 418.683,Z 395.302,A -85,B 0,C 180,E1 -10600.562,E2 -10600.562} C_VEL
LIN {X 0,Y 419.027,Z 399.449,A -85,B 0,C 180,E1 -10600.698,E2 -10600.698} C_VEL
LIN {X 0,Y 416.612,Z 481.39,A -85,B 0,C 180,E1 -10602.608,E2 -10602.608} C_VEL
LIN {X 0,Y 416.214,Z 495.237,A -85,B 0,C 180,E1 -10603.003,E2 -10603.003} C_VEL
LIN {X 0,Y 415.676,Z 507.847,A -85,B 0,C 180,E1 -10603.549,E2 -10603.549} C_VEL
LIN {X 0,Y 415.106,Z 520.127,A -85,B 0,C 180,E1 -10604.283,E2 -10604.283} C_VEL
LIN {X 0,Y 414.331,Z 532.151,A -85,B 0,C 180,E1 -10605.209,E2 -10605.209} C_VEL
LIN {X 0,Y 413.552,Z 543.766,A -85,B 0,C 180,E1 -10606.362,E2 -10606.362} C_VEL
LIN {X 0,Y 412.804,Z 552.838,A -85,B 0,C 180,E1 -10607.463,E2 -10607.463} C_VEL
LIN {X 0,Y 412.206,Z 561.104,A -85,B 0,C 180,E1 -10608.693,E2 -10608.693} C_VEL
LIN {X 0,Y 411.607,Z 569.156,A -85,B 0,C 180,E1 -10610.169,E2 -10610.169} C_VEL
LIN {X 0,Y 411.052,Z 575.652,A -85,B 0,C 180,E1 -10611.644,E2 -10611.644} C_VEL
LIN {X 0,Y 410.715,Z 580.769,A -85,B 0,C 180,E1 -10613.121,E2 -10613.121} C_VEL
LIN {X 0,Y 410.326,Z 584.685,A -85,B 0,C 180,E1 -10614.595,E2 -10614.595} C_VEL
LIN {X 0,Y 410.336,Z 587.502,A -85,B 0,C 180,E1 -10616.072,E2 -10616.072} C_VEL
LIN {X 0,Y 410.197,Z 588.816,A -85,B 0,C 180,E1 -10617.054,E2 -10617.054} C_VEL
LIN {X 0,Y 410.075,Z 589.72,A -85,B 0,C 180,E1 -10618.036,E2 -10618.036} C_VEL
LIN {X 0,Y 410.008,Z 590.198,A -85,B 0,C 180,E1 -10619.018,E2 -10619.018} C_VEL
LIN {X 0,Y 409.975,Z 590.211,A -85,B 0,C 180,E1 -10620,E2 -10620} C_VEL
LIN {X 0,Y 409.985,Z 589.816,A -85,B 0,C 180,E1 -10620.982,E2 -10620.982} C_VEL
LIN {X 0,Y 410.054,Z 589.009,A -85,B 0,C 180,E1 -10621.964,E2 -10621.964} C_VEL
LIN {X 0,Y 410.145,Z 587.729,A -85,B 0,C 180,E1 -10622.947,E2 -10622.947} C_VEL
LIN {X 0,Y 410.14,Z 585.006,A -85,B 0,C 180,E1 -10624.423,E2 -10624.423} C_VEL
LIN {X 0,Y 410.348,Z 581.207,A -85,B 0,C 180,E1 -10625.898,E2 -10625.898} C_VEL
LIN {X 0,Y 410.532,Z 576.233,A -85,B 0,C 180,E1 -10627.377,E2 -10627.377} C_VEL
LIN {X 0,Y 410.839,Z 569.942,A -85,B 0,C 180,E1 -10628.856,E2 -10628.856} C_VEL
LIN {X 0,Y 411.296,Z 562.05,A -85,B 0,C 180,E1 -10630.336,E2 -10630.336} C_VEL
LIN {X 0,Y 411.869,Z 552.185,A -85,B 0,C 180,E1 -10631.816,E2 -10631.816} C_VEL
LIN {X 0,Y 412.533,Z 541.906,A -85,B 0,C 180,E1 -10633.046,E2 -10633.046} C_VEL
LIN {X 0,Y 413.067,Z 530.33,A -85,B 0,C 180,E1 -10634.165,E2 -10634.165} C_VEL
LIN {X 0,Y 413.588,Z 519.082,A -85,B 0,C 180,E1 -10635.019,E2 -10635.019} C_VEL
LIN {X 0,Y 414.129,Z 506.54,A -85,B 0,C 180,E1 -10635.755,E2 -10635.755} C_VEL
LIN {X 0,Y 414.549,Z 493.601,A -85,B 0,C 180,E1 -10636.308,E2 -10636.308} C_VEL
LIN {X 0,Y 414.865,Z 478.761,A -85,B 0,C 180,E1 -10636.706,E2 -10636.706} C_VEL
LIN {X 0,Y 416.303,Z 396.127,A -85,B 0,C 180,E1 -10638.426,E2 -10638.426} C_VEL
LIN {X 0,Y 413.19,Z 377.33,A -85,B 0,C 180,E1 -10638.984,E2 -10638.984} C_VEL
LIN {X 0,Y 413.897,Z 358.332,A -85,B 0,C 180,E1 -10642.461,E2 -10642.461} C_VEL
LIN {X 0,Y 413.166,Z 352.327,A -85,B 0,C 180,E1 -10643.61,E2 -10643.61} C_VEL
LIN {X 0,Y 411.26,Z 342.883,A -85,B 0,C 180,E1 -10645.495,E2 -10645.495} C_VEL
LIN {X 0,Y 411.224,Z 342.886,A -85,B 0,C 180,E1 -10648.59,E2 -10648.59} C_VEL
LIN {X 0,Y 411.172,Z 342.893,A -85,B 0,C 180,E1 -10651.997,E2 -10651.997} C_VEL
LIN {X 0,Y 411.216,Z 342.885,A -85,B 0,C 180,E1 -10654.878,E2 -10654.878} C_VEL
LIN {X 0,Y 411.2,Z 342.889,A -85,B 0,C 180,E1 -10658.166,E2 -10658.166} C_VEL
LIN {X 0,Y 411.175,Z 342.896,A -85,B 0,C 180,E1 -10661.806,E2 -10661.806} C_VEL
LIN {X 0,Y 411.18,Z 342.893,A -85,B 0,C 180,E1 -10665.509,E2 -10665.509} C_VEL
LIN {X 0,Y 411.154,Z 342.893,A -85,B 0,C 180,E1 -10668.774,E2 -10668.774} C_VEL
LIN {X 0,Y 411.187,Z 342.892,A -85,B 0,C 180,E1 -10672.024,E2 -10672.024} C_VEL
LIN {X 0,Y 411.207,Z 342.886,A -85,B 0,C 180,E1 -10675.123,E2 -10675.123} C_VEL
LIN {X 0,Y 411.159,Z 342.896,A -85,B 0,C 180,E1 -10678.001,E2 -10678.001} C_VEL
LIN {X 0,Y 411.191,Z 342.893,A -85,B 0,C 180,E1 -10681.407,E2 -10681.407} C_VEL
LIN {X 0,Y 411.24,Z 343.045,A -85,B 0,C 180,E1 -10681.932,E2 -10681.932} C_VEL
LIN {X 0,Y 414.02,Z 355.918,A -85,B 0,C 180,E1 -10684.888,E2 -10684.888} C_VEL
LIN {X 0,Y 415.169,Z 362.247,A -85,B 0,C 180,E1 -10686.282,E2 -10686.282} C_VEL
LIN {X 0,Y 415.096,Z 363.657,A -85,B 0,C 180,E1 -10686.57,E2 -10686.57} C_VEL
LIN {X 0,Y 420.547,Z 390.155,A -85,B 0,C 180,E1 -10687.379,E2 -10687.379} C_VEL
LIN {X 0,Y 419.107,Z 489.35,A -85,B 0,C 180,E1 -10689.091,E2 -10689.091} C_VEL
LIN {X 0,Y 418.7,Z 505.109,A -85,B 0,C 180,E1 -10689.423,E2 -10689.423} C_VEL
LIN {X 0,Y 418.048,Z 519.055,A -85,B 0,C 180,E1 -10689.903,E2 -10689.903} C_VEL
LIN {X 0,Y 417.82,Z 524.744,A -85,B 0,C 180,E1 -10690.164,E2 -10690.164} C_VEL
LIN {X 0,Y 416.878,Z 530.308,A -85,B 0,C 180,E1 -10690.411,E2 -10690.411} C_VEL
LIN {X 0,Y 413.537,Z 539.232,A -85,B 0,C 180,E1 -10690.803,E2 -10690.803} C_VEL
LIN {X 0,Y 410.164,Z 547.853,A -85,B 0,C 180,E1 -10691.291,E2 -10691.291} C_VEL
LIN {X 0,Y 409.175,Z 552.934,A -85,B 0,C 180,E1 -10691.684,E2 -10691.684} C_VEL
LIN {X 0,Y 407.956,Z 565.163,A -85,B 0,C 180,E1 -10692.84,E2 -10692.84} C_VEL
LIN {X 0,Y 406.851,Z 576.853,A -85,B 0,C 180,E1 -10694.211,E2 -10694.211} C_VEL
LIN {X 0,Y 405.764,Z 587.296,A -85,B 0,C 180,E1 -10695.709,E2 -10695.709} C_VEL
LIN {X 0,Y 405.03,Z 595.908,A -85,B 0,C 180,E1 -10697.217,E2 -10697.217} C_VEL
LIN {X 0,Y 404.144,Z 604.165,A -85,B 0,C 180,E1 -10698.971,E2 -10698.971} C_VEL
LIN {X 0,Y 403.676,Z 609.919,A -85,B 0,C 180,E1 -10700.478,E2 -10700.478} C_VEL
LIN {X 0,Y 403.313,Z 614.65,A -85,B 0,C 180,E1 -10701.985,E2 -10701.985} C_VEL
LIN {X 0,Y 403.067,Z 619.545,A -85,B 0,C 180,E1 -10703.993,E2 -10703.993} C_VEL
LIN {X 0,Y 402.866,Z 622.957,A -85,B 0,C 180,E1 -10705.997,E2 -10705.997} C_VEL
LIN {X 0,Y 402.864,Z 624.986,A -85,B 0,C 180,E1 -10707.999,E2 -10707.999} C_VEL
LIN {X 0,Y 402.831,Z 625.686,A -85,B 0,C 180,E1 -10709.998,E2 -10709.998} C_VEL
LIN {X 0,Y 402.863,Z 625.062,A -85,B 0,C 180,E1 -10711.998,E2 -10711.998} C_VEL
LIN {X 0,Y 402.864,Z 623.104,A -85,B 0,C 180,E1 -10714,E2 -10714} C_VEL
LIN {X 0,Y 403.023,Z 619.758,A -85,B 0,C 180,E1 -10716.004,E2 -10716.004} C_VEL
LIN {X 0,Y 403.308,Z 614.928,A -85,B 0,C 180,E1 -10718.012,E2 -10718.012} C_VEL
LIN {X 0,Y 403.818,Z 608.468,A -85,B 0,C 180,E1 -10720.021,E2 -10720.021} C_VEL
LIN {X 0,Y 404.476,Z 601.274,A -85,B 0,C 180,E1 -10721.779,E2 -10721.779} C_VEL
LIN {X 0,Y 405.243,Z 593.32,A -85,B 0,C 180,E1 -10723.361,E2 -10723.361} C_VEL
LIN {X 0,Y 406.033,Z 584.682,A -85,B 0,C 180,E1 -10724.79,E2 -10724.79} C_VEL
LIN {X 0,Y 407.188,Z 573.712,A -85,B 0,C 180,E1 -10726.287,E2 -10726.287} C_VEL
LIN {X 0,Y 408.292,Z 562.531,A -85,B 0,C 180,E1 -10727.53,E2 -10727.53} C_VEL
LIN {X 0,Y 409.411,Z 550.161,A -85,B 0,C 180,E1 -10728.644,E2 -10728.644} C_VEL
LIN {X 0,Y 410.33,Z 537.686,A -85,B 0,C 180,E1 -10729.546,E2 -10729.546} C_VEL
LIN {X 0,Y 411.223,Z 523.896,A -85,B 0,C 180,E1 -10730.311,E2 -10730.311} C_VEL
LIN {X 0,Y 411.926,Z 509.306,A -85,B 0,C 180,E1 -10730.895,E2 -10730.895} C_VEL
LIN {X 0,Y 412.441,Z 494.802,A -85,B 0,C 180,E1 -10731.26,E2 -10731.26} C_VEL
LIN {X 0,Y 414.003,Z 390.952,A -85,B 0,C 180,E1 -10733.084,E2 -10733.084} C_VEL
LIN {X 0,Y 408.421,Z 364.505,A -85,B 0,C 180,E1 -10733.917,E2 -10733.917} C_VEL
LIN {X 0,Y 408.262,Z 363.596,A -85,B 0,C 180,E1 -10733.974,E2 -10733.974} C_VEL
LIN {X 0,Y 406.12,Z 352.518,A -85,B 0,C 180,E1 -10736.489,E2 -10736.489} C_VEL
LIN {X 0,Y 404.161,Z 343.771,A -85,B 0,C 180,E1 -10738.566,E2 -10738.566} C_VEL
LIN {X 0,Y 404.132,Z 343.774,A -85,B 0,C 180,E1 -10741.556,E2 -10741.556} C_VEL
LIN {X 0,Y 404.176,Z 343.768,A -85,B 0,C 180,E1 -10745.015,E2 -10745.015} C_VEL
LIN {X 0,Y 404.126,Z 343.773,A -85,B 0,C 180,E1 -10748.758,E2 -10748.758} C_VEL
LIN {X 0,Y 404.097,Z 343.772,A -85,B 0,C 180,E1 -10751.595,E2 -10751.595} C_VEL
LIN {X 0,Y 404.134,Z 343.769,A -85,B 0,C 180,E1 -10754.52,E2 -10754.52} C_VEL
LIN {X 0,Y 404.112,Z 343.772,A -85,B 0,C 180,E1 -10757.292,E2 -10757.292} C_VEL
LIN {X 0,Y 404.122,Z 343.769,A -85,B 0,C 180,E1 -10759.95,E2 -10759.95} C_VEL
LIN {X 0,Y 404.123,Z 343.769,A -85,B 0,C 180,E1 -10763.124,E2 -10763.124} C_VEL
LIN {X 0,Y 404.126,Z 343.766,A -85,B 0,C 180,E1 -10766.186,E2 -10766.186} C_VEL
LIN {X 0,Y 404.13,Z 343.767,A -85,B 0,C 180,E1 -10769.713,E2 -10769.713} C_VEL
LIN {X 0,Y 404.091,Z 343.759,A -85,B 0,C 180,E1 -10773.115,E2 -10773.115} C_VEL
LIN {X 0,Y 404.135,Z 343.768,A -85,B 0,C 180,E1 -10776.423,E2 -10776.423} C_VEL
LIN {X 0,Y 404.178,Z 343.751,A -85,B 0,C 180,E1 -10779.874,E2 -10779.874} C_VEL
LIN {X 0,Y 404.202,Z 343.759,A -85,B 0,C 180,E1 -10782.992,E2 -10782.992} C_VEL
LIN {X 0,Y 404.269,Z 343.75,A -85,B 0,C 180,E1 -10786.938,E2 -10786.938} C_VEL
LIN {X 0,Y 404.239,Z 343.754,A -85,B 0,C 180,E1 -10789.988,E2 -10789.988} C_VEL
LIN {X 0,Y 404.321,Z 343.746,A -85,B 0,C 180,E1 -10793.011,E2 -10793.011} C_VEL
LIN {X 0,Y 404.242,Z 343.75,A -85,B 0,C 180,E1 -10795.013,E2 -10795.013} C_VEL
LIN {X 0,Y 404.459,Z 343.727,A -85,B 0,C 180,E1 -10798.008,E2 -10798.008} C_VEL
LIN {X 0,Y 404.456,Z 343.727,A -85,B 0,C 180,E1 -10801.992,E2 -10801.992} C_VEL
LIN {X 0,Y 404.364,Z 343.738,A -85,B 0,C 180,E1 -10805.986,E2 -10805.986} C_VEL
LIN {X 0,Y 404.24,Z 343.753,A -85,B 0,C 180,E1 -10809.002,E2 -10809.002} C_VEL
LIN {X 0,Y 404.233,Z 343.756,A -85,B 0,C 180,E1 -10812.042,E2 -10812.042} C_VEL
LIN {X 0,Y 404.19,Z 343.759,A -85,B 0,C 180,E1 -10815.119,E2 -10815.119} C_VEL
LIN {X 0,Y 404.189,Z 343.762,A -85,B 0,C 180,E1 -10818.239,E2 -10818.239} C_VEL
LIN {X 0,Y 404.123,Z 343.758,A -85,B 0,C 180,E1 -10821.42,E2 -10821.42} C_VEL
LIN {X 0,Y 404.121,Z 343.772,A -85,B 0,C 180,E1 -10824.669,E2 -10824.669} C_VEL
LIN {X 0,Y 404.092,Z 343.768,A -85,B 0,C 180,E1 -10828.007,E2 -10828.007} C_VEL
LIN {X 0,Y 404.129,Z 343.763,A -85,B 0,C 180,E1 -10830.286,E2 -10830.286} C_VEL
LIN {X 0,Y 404.125,Z 343.767,A -85,B 0,C 180,E1 -10833.814,E2 -10833.814} C_VEL
LIN {X 0,Y 404.118,Z 343.771,A -85,B 0,C 180,E1 -10836.875,E2 -10836.875} C_VEL
LIN {X 0,Y 404.105,Z 343.775,A -85,B 0,C 180,E1 -10840.076,E2 -10840.076} C_VEL
LIN {X 0,Y 404.129,Z 343.767,A -85,B 0,C 180,E1 -10843.083,E2 -10843.083} C_VEL
LIN {X 0,Y 404.109,Z 343.773,A -85,B 0,C 180,E1 -10845.923,E2 -10845.923} C_VEL
LIN {X 0,Y 404.09,Z 343.777,A -85,B 0,C 180,E1 -10848.634,E2 -10848.634} C_VEL
LIN {X 0,Y 404.124,Z 343.771,A -85,B 0,C 180,E1 -10851.498,E2 -10851.498} C_VEL
LIN {X 0,Y 404.164,Z 343.766,A -85,B 0,C 180,E1 -10854.984,E2 -10854.984} C_VEL
LIN {X 0,Y 404.13,Z 343.772,A -85,B 0,C 180,E1 -10858.444,E2 -10858.444} C_VEL
LIN {X 0,Y 404.167,Z 343.857,A -85,B 0,C 180,E1 -10860.277,E2 -10860.277} C_VEL
LIN {X 0,Y 406.912,Z 356.037,A -85,B 0,C 180,E1 -10863.041,E2 -10863.041} C_VEL
LIN {X 0,Y 408.56,Z 364.094,A -85,B 0,C 180,E1 -10864.804,E2 -10864.804} C_VEL
LIN {X 0,Y 408.223,Z 370.845,A -85,B 0,C 180,E1 -10866.102,E2 -10866.102} C_VEL
LIN {X 0,Y 413.873,Z 399.607,A -85,B 0,C 180,E1 -10866.98,E2 -10866.98} C_VEL
LIN {X 0,Y 412.226,Z 507.521,A -85,B 0,C 180,E1 -10868.892,E2 -10868.892} C_VEL
LIN {X 0,Y 411.623,Z 521.628,A -85,B 0,C 180,E1 -10869.318,E2 -10869.318} C_VEL
LIN {X 0,Y 410.819,Z 535.319,A -85,B 0,C 180,E1 -10869.929,E2 -10869.929} C_VEL
LIN {X 0,Y 409.952,Z 548.236,A -85,B 0,C 180,E1 -10870.705,E2 -10870.705} C_VEL
LIN {X 0,Y 408.971,Z 559.988,A -85,B 0,C 180,E1 -10871.595,E2 -10871.595} C_VEL
LIN {X 0,Y 407.851,Z 571.873,A -85,B 0,C 180,E1 -10872.709,E2 -10872.709} C_VEL
LIN {X 0,Y 406.793,Z 582.732,A -85,B 0,C 180,E1 -10873.955,E2 -10873.955} C_VEL
LIN {X 0,Y 405.69,Z 593.463,A -85,B 0,C 180,E1 -10875.454,E2 -10875.454} C_VEL
LIN {X 0,Y 404.869,Z 602.323,A -85,B 0,C 180,E1 -10876.96,E2 -10876.96} C_VEL
LIN {X 0,Y 404.227,Z 609.696,A -85,B 0,C 180,E1 -10878.468,E2 -10878.468} C_VEL
LIN {X 0,Y 403.662,Z 615.841,A -85,B 0,C 180,E1 -10879.975,E2 -10879.975} C_VEL
LIN {X 0,Y 403.192,Z 622.367,A -85,B 0,C 180,E1 -10881.986,E2 -10881.986} C_VEL
LIN {X 0,Y 402.985,Z 627.257,A -85,B 0,C 180,E1 -10883.995,E2 -10883.995} C_VEL
LIN {X 0,Y 402.831,Z 630.654,A -85,B 0,C 180,E1 -10886,E2 -10886} C_VEL
LIN {X 0,Y 402.819,Z 632.659,A -85,B 0,C 180,E1 -10888.002,E2 -10888.002} C_VEL
LIN {X 0,Y 402.83,Z 633.321,A -85,B 0,C 180,E1 -10890.002,E2 -10890.002} C_VEL
LIN {X 0,Y 402.82,Z 632.651,A -85,B 0,C 180,E1 -10892.001,E2 -10892.001} C_VEL
LIN {X 0,Y 402.83,Z 630.637,A -85,B 0,C 180,E1 -10894.003,E2 -10894.003} C_VEL
LIN {X 0,Y 402.987,Z 627.236,A -85,B 0,C 180,E1 -10896.008,E2 -10896.008} C_VEL
LIN {X 0,Y 403.195,Z 622.344,A -85,B 0,C 180,E1 -10898.017,E2 -10898.017} C_VEL
LIN {X 0,Y 403.665,Z 615.808,A -85,B 0,C 180,E1 -10900.028,E2 -10900.028} C_VEL
LIN {X 0,Y 404.351,Z 608.536,A -85,B 0,C 180,E1 -10901.786,E2 -10901.786} C_VEL
LIN {X 0,Y 405.119,Z 599.541,A -85,B 0,C 180,E1 -10903.544,E2 -10903.544} C_VEL
LIN {X 0,Y 406.038,Z 590.078,A -85,B 0,C 180,E1 -10905.049,E2 -10905.049} C_VEL
LIN {X 0,Y 407.114,Z 579.616,A -85,B 0,C 180,E1 -10906.422,E2 -10906.422} C_VEL
LIN {X 0,Y 408.208,Z 568.065,A -85,B 0,C 180,E1 -10907.666,E2 -10907.666} C_VEL
LIN {X 0,Y 409.367,Z 555.249,A -85,B 0,C 180,E1 -10908.779,E2 -10908.779} C_VEL
LIN {X 0,Y 410.433,Z 541.765,A -85,B 0,C 180,E1 -10909.701,E2 -10909.701} C_VEL
LIN {X 0,Y 411.162,Z 528.805,A -85,B 0,C 180,E1 -10910.383,E2 -10910.383} C_VEL
LIN {X 0,Y 411.932,Z 515.044,A -85,B 0,C 180,E1 -10910.898,E2 -10910.898} C_VEL
LIN {X 0,Y 412.318,Z 500.975,A -85,B 0,C 180,E1 -10911.237,E2 -10911.237} C_VEL
LIN {X 0,Y 413.883,Z 402.721,A -85,B 0,C 180,E1 -10912.954,E2 -10912.954} C_VEL
LIN {X 0,Y 413.571,Z 397.889,A -85,B 0,C 180,E1 -10913.062,E2 -10913.062} C_VEL
LIN {X 0,Y 408.141,Z 370.458,A -85,B 0,C 180,E1 -10913.924,E2 -10913.924} C_VEL
LIN {X 0,Y 408.548,Z 364.028,A -85,B 0,C 180,E1 -10915.2,E2 -10915.2} C_VEL
LIN {X 0,Y 405.735,Z 350.591,A -85,B 0,C 180,E1 -10918.166,E2 -10918.166} C_VEL
LIN {X 0,Y 404.166,Z 343.765,A -85,B 0,C 180,E1 -10919.751,E2 -10919.751} C_VEL
LIN {X 0,Y 404.176,Z 343.764,A -85,B 0,C 180,E1 -10923.421,E2 -10923.421} C_VEL
LIN {X 0,Y 404.146,Z 343.766,A -85,B 0,C 180,E1 -10926.247,E2 -10926.247} C_VEL
LIN {X 0,Y 404.157,Z 343.763,A -85,B 0,C 180,E1 -10928.758,E2 -10928.758} C_VEL
LIN {X 0,Y 404.128,Z 343.769,A -85,B 0,C 180,E1 -10931.6,E2 -10931.6} C_VEL
LIN {X 0,Y 404.15,Z 343.766,A -85,B 0,C 180,E1 -10934.523,E2 -10934.523} C_VEL
LIN {X 0,Y 404.142,Z 343.769,A -85,B 0,C 180,E1 -10937.296,E2 -10937.296} C_VEL
LIN {X 0,Y 404.174,Z 343.762,A -85,B 0,C 180,E1 -10939.956,E2 -10939.956} C_VEL
LIN {X 0,Y 404.141,Z 343.767,A -85,B 0,C 180,E1 -10943.126,E2 -10943.126} C_VEL
LIN {X 0,Y 404.15,Z 343.769,A -85,B 0,C 180,E1 -10946.188,E2 -10946.188} C_VEL
LIN {X 0,Y 404.15,Z 343.772,A -85,B 0,C 180,E1 -10949.715,E2 -10949.715} C_VEL
LIN {X 0,Y 404.204,Z 343.892,A -85,B 0,C 180,E1 -10951.86,E2 -10951.86} C_VEL
LIN {X 0,Y 407.547,Z 355.356,A -85,B 0,C 180,E1 -10954.462,E2 -10954.462} C_VEL
LIN {X 0,Y 409.316,Z 364.258,A -85,B 0,C 180,E1 -10956.318,E2 -10956.318} C_VEL
LIN {X 0,Y 409.089,Z 373.698,A -85,B 0,C 180,E1 -10958.081,E2 -10958.081} C_VEL
LIN {X 0,Y 408.783,Z 380.975,A -85,B 0,C 180,E1 -10959.411,E2 -10959.411} C_VEL
LIN {X 0,Y 412.238,Z 395.922,A -85,B 0,C 180,E1 -10960.11,E2 -10960.11} C_VEL
LIN {X 0,Y 412.723,Z 399.595,A -85,B 0,C 180,E1 -10960.25,E2 -10960.25} C_VEL
LIN {X 0,Y 410.113,Z 478.832,A -85,B 0,C 180,E1 -10962.162,E2 -10962.162} C_VEL
LIN {X 0,Y 409.709,Z 493.5,A -85,B 0,C 180,E1 -10962.563,E2 -10962.563} C_VEL
LIN {X 0,Y 409.13,Z 507.309,A -85,B 0,C 180,E1 -10963.149,E2 -10963.149} C_VEL
LIN {X 0,Y 408.498,Z 519.754,A -85,B 0,C 180,E1 -10963.894,E2 -10963.894} C_VEL
LIN {X 0,Y 407.693,Z 531.348,A -85,B 0,C 180,E1 -10964.784,E2 -10964.784} C_VEL
LIN {X 0,Y 406.951,Z 542.11,A -85,B 0,C 180,E1 -10965.835,E2 -10965.835} C_VEL
LIN {X 0,Y 406.073,Z 551.842,A -85,B 0,C 180,E1 -10966.998,E2 -10966.998} C_VEL
LIN {X 0,Y 405.425,Z 560.36,A -85,B 0,C 180,E1 -10968.248,E2 -10968.248} C_VEL
LIN {X 0,Y 404.736,Z 568.643,A -85,B 0,C 180,E1 -10969.748,E2 -10969.748} C_VEL
LIN {X 0,Y 404.196,Z 574.299,A -85,B 0,C 180,E1 -10970.997,E2 -10970.997} C_VEL
LIN {X 0,Y 403.776,Z 579.77,A -85,B 0,C 180,E1 -10972.5,E2 -10972.5} C_VEL
LIN {X 0,Y 403.446,Z 584.009,A -85,B 0,C 180,E1 -10974.001,E2 -10974.001} C_VEL
LIN {X 0,Y 403.209,Z 586.241,A -85,B 0,C 180,E1 -10975,E2 -10975} C_VEL
LIN {X 0,Y 403.28,Z 587.962,A -85,B 0,C 180,E1 -10976.003,E2 -10976.003} C_VEL
LIN {X 0,Y 403.14,Z 589.249,A -85,B 0,C 180,E1 -10977.002,E2 -10977.002} C_VEL
LIN {X 0,Y 403.007,Z 590.127,A -85,B 0,C 180,E1 -10978.001,E2 -10978.001} C_VEL
LIN {X 0,Y 402.932,Z 590.555,A -85,B 0,C 180,E1 -10979.001,E2 -10979.001} C_VEL
LIN {X 0,Y 402.898,Z 590.538,A -85,B 0,C 180,E1 -10980,E2 -10980} C_VEL
LIN {X 0,Y 402.91,Z 590.113,A -85,B 0,C 180,E1 -10981,E2 -10981} C_VEL
LIN {X 0,Y 402.986,Z 589.257,A -85,B 0,C 180,E1 -10981.999,E2 -10981.999} C_VEL
LIN {X 0,Y 403.048,Z 587.938,A -85,B 0,C 180,E1 -10982.999,E2 -10982.999} C_VEL
LIN {X 0,Y 403.066,Z 585.146,A -85,B 0,C 180,E1 -10984.5,E2 -10984.5} C_VEL
LIN {X 0,Y 403.266,Z 581.271,A -85,B 0,C 180,E1 -10986.002,E2 -10986.002} C_VEL
LIN {X 0,Y 403.482,Z 576.214,A -85,B 0,C 180,E1 -10987.507,E2 -10987.507} C_VEL
LIN {X 0,Y 403.815,Z 569.826,A -85,B 0,C 180,E1 -10989.012,E2 -10989.012} C_VEL
LIN {X 0,Y 404.286,Z 561.786,A -85,B 0,C 180,E1 -10990.517,E2 -10990.517} C_VEL
LIN {X 0,Y 404.746,Z 553.58,A -85,B 0,C 180,E1 -10991.773,E2 -10991.773} C_VEL
LIN {X 0,Y 405.415,Z 543.604,A -85,B 0,C 180,E1 -10993.024,E2 -10993.024} C_VEL
LIN {X 0,Y 405.955,Z 532.648,A -85,B 0,C 180,E1 -10994.13,E2 -10994.13} C_VEL
LIN {X 0,Y 406.516,Z 521.542,A -85,B 0,C 180,E1 -10995.03,E2 -10995.03} C_VEL
LIN {X 0,Y 407.028,Z 509.697,A -85,B 0,C 180,E1 -10995.78,E2 -10995.78} C_VEL
LIN {X 0,Y 407.546,Z 495.543,A -85,B 0,C 180,E1 -10996.435,E2 -10996.435} C_VEL
LIN {X 0,Y 407.865,Z 481.949,A -85,B 0,C 180,E1 -10996.84,E2 -10996.84} C_VEL
LIN {X 0,Y 409.362,Z 396.421,A -85,B 0,C 180,E1 -10998.676,E2 -10998.676} C_VEL
LIN {X 0,Y 406.256,Z 377.691,A -85,B 0,C 180,E1 -10999.222,E2 -10999.222} C_VEL
LIN {X 0,Y 406.953,Z 359.402,A -85,B 0,C 180,E1 -11002.598,E2 -11002.598} C_VEL
LIN {X 0,Y 405.95,Z 352.417,A -85,B 0,C 180,E1 -11003.953,E2 -11003.953} C_VEL
LIN {X 0,Y 404.238,Z 343.758,A -85,B 0,C 180,E1 -11005.697,E2 -11005.697} C_VEL
LIN {X 0,Y 404.202,Z 343.764,A -85,B 0,C 180,E1 -11007.999,E2 -11007.999} C_VEL
LIN {X 0,Y 404.145,Z 343.764,A -85,B 0,C 180,E1 -11011.558,E2 -11011.558} C_VEL
LIN {X 0,Y 404.19,Z 343.76,A -85,B 0,C 180,E1 -11015.016,E2 -11015.016} C_VEL
LIN {X 0,Y 404.14,Z 343.766,A -85,B 0,C 180,E1 -11018.759,E2 -11018.759} C_VEL
LIN {X 0,Y 404.119,Z 343.772,A -85,B 0,C 180,E1 -11021.598,E2 -11021.598} C_VEL
LIN {X 0,Y 404.151,Z 343.766,A -85,B 0,C 180,E1 -11024.521,E2 -11024.521} C_VEL
LIN {X 0,Y 404.13,Z 343.771,A -85,B 0,C 180,E1 -11027.293,E2 -11027.293} C_VEL
LIN {X 0,Y 404.138,Z 343.769,A -85,B 0,C 180,E1 -11029.95,E2 -11029.95} C_VEL
LIN {X 0,Y 404.137,Z 343.771,A -85,B 0,C 180,E1 -11033.125,E2 -11033.125} C_VEL
LIN {X 0,Y 404.142,Z 343.769,A -85,B 0,C 180,E1 -11036.186,E2 -11036.186} C_VEL
LIN {X 0,Y 404.145,Z 343.768,A -85,B 0,C 180,E1 -11039.714,E2 -11039.714} C_VEL
LIN {X 0,Y 404.198,Z 343.904,A -85,B 0,C 180,E1 -11041.575,E2 -11041.575} C_VEL
LIN {X 0,Y 407.091,Z 357.265,A -85,B 0,C 180,E1 -11044.703,E2 -11044.703} C_VEL
LIN {X 0,Y 408.292,Z 363.705,A -85,B 0,C 180,E1 -11046.151,E2 -11046.151} C_VEL
LIN {X 0,Y 413.85,Z 390.13,A -85,B 0,C 180,E1 -11046.99,E2 -11046.99} C_VEL
LIN {X 0,Y 413.794,Z 408.855,A -85,B 0,C 180,E1 -11047.332,E2 -11047.332} C_VEL
LIN {X 0,Y 412.241,Z 500.618,A -85,B 0,C 180,E1 -11048.955,E2 -11048.955} C_VEL
LIN {X 0,Y 411.666,Z 515.324,A -85,B 0,C 180,E1 -11049.415,E2 -11049.415} C_VEL
LIN {X 0,Y 410.959,Z 528.182,A -85,B 0,C 180,E1 -11049.998,E2 -11049.998} C_VEL
LIN {X 0,Y 410.157,Z 540.495,A -85,B 0,C 180,E1 -11050.737,E2 -11050.737} C_VEL
LIN {X 0,Y 409.175,Z 552.934,A -85,B 0,C 180,E1 -11051.684,E2 -11051.684} C_VEL
LIN {X 0,Y 408.176,Z 557.996,A -85,B 0,C 180,E1 -11052.106,E2 -11052.106} C_VEL
LIN {X 0,Y 404.662,Z 565.959,A -85,B 0,C 180,E1 -11052.781,E2 -11052.781} C_VEL
LIN {X 0,Y 401.063,Z 573.518,A -85,B 0,C 180,E1 -11053.522,E2 -11053.522} C_VEL
LIN {X 0,Y 399.899,Z 577.879,A -85,B 0,C 180,E1 -11054.06,E2 -11054.06} C_VEL
LIN {X 0,Y 398.853,Z 587.367,A -85,B 0,C 180,E1 -11055.456,E2 -11055.456} C_VEL
LIN {X 0,Y 398.086,Z 595.978,A -85,B 0,C 180,E1 -11056.99,E2 -11056.99} C_VEL
LIN {X 0,Y 397.139,Z 604.234,A -85,B 0,C 180,E1 -11058.774,E2 -11058.774} C_VEL
LIN {X 0,Y 396.65,Z 609.988,A -85,B 0,C 180,E1 -11060.308,E2 -11060.308} C_VEL
LIN {X 0,Y 396.254,Z 614.719,A -85,B 0,C 180,E1 -11061.841,E2 -11061.841} C_VEL
LIN {X 0,Y 395.999,Z 619.614,A -85,B 0,C 180,E1 -11063.886,E2 -11063.886} C_VEL
LIN {X 0,Y 395.791,Z 623.025,A -85,B 0,C 180,E1 -11065.926,E2 -11065.926} C_VEL
LIN {X 0,Y 395.762,Z 625.054,A -85,B 0,C 180,E1 -11067.963,E2 -11067.963} C_VEL
LIN {X 0,Y 395.759,Z 625.753,A -85,B 0,C 180,E1 -11069.998,E2 -11069.998} C_VEL
LIN {X 0,Y 395.761,Z 625.129,A -85,B 0,C 180,E1 -11072.034,E2 -11072.034} C_VEL
LIN {X 0,Y 395.789,Z 623.17,A -85,B 0,C 180,E1 -11074.071,E2 -11074.071} C_VEL
LIN {X 0,Y 395.949,Z 619.825,A -85,B 0,C 180,E1 -11076.112,E2 -11076.112} C_VEL
LIN {X 0,Y 396.249,Z 614.994,A -85,B 0,C 180,E1 -11078.156,E2 -11078.156} C_VEL
LIN {X 0,Y 396.808,Z 608.533,A -85,B 0,C 180,E1 -11080.2,E2 -11080.2} C_VEL
LIN {X 0,Y 397.513,Z 601.34,A -85,B 0,C 180,E1 -11081.988,E2 -11081.988} C_VEL
LIN {X 0,Y 398.255,Z 593.64,A -85,B 0,C 180,E1 -11083.551,E2 -11083.551} C_VEL
LIN {X 0,Y 399.15,Z 584.746,A -85,B 0,C 180,E1 -11085.051,E2 -11085.051} C_VEL
LIN {X 0,Y 400.318,Z 573.777,A -85,B 0,C 180,E1 -11086.574,E2 -11086.574} C_VEL
LIN {X 0,Y 401.487,Z 562.595,A -85,B 0,C 180,E1 -11087.837,E2 -11087.837} C_VEL
LIN {X 0,Y 402.673,Z 550.223,A -85,B 0,C 180,E1 -11088.968,E2 -11088.968} C_VEL
LIN {X 0,Y 403.672,Z 537.129,A -85,B 0,C 180,E1 -11089.923,E2 -11089.923} C_VEL
LIN {X 0,Y 404.623,Z 522.655,A -85,B 0,C 180,E1 -11090.724,E2 -11090.724} C_VEL
LIN {X 0,Y 405.325,Z 508.446,A -85,B 0,C 180,E1 -11091.285,E2 -11091.285} C_VEL
LIN {X 0,Y 405.847,Z 494.847,A -85,B 0,C 180,E1 -11091.623,E2 -11091.623} C_VEL
LIN {X 0,Y 407.514,Z 392.513,A -85,B 0,C 180,E1 -11093.445,E2 -11093.445} C_VEL
LIN {X 0,Y 402.595,Z 368.595,A -85,B 0,C 180,E1 -11094.207,E2 -11094.207} C_VEL
LIN {X 0,Y 401.202,Z 363.7,A -85,B 0,C 180,E1 -11094.415,E2 -11094.415} C_VEL
LIN {X 0,Y 398.403,Z 350.377,A -85,B 0,C 180,E1 -11097.536,E2 -11097.536} C_VEL
LIN {X 0,Y 397.13,Z 344.646,A -85,B 0,C 180,E1 -11098.975,E2 -11098.975} C_VEL
LIN {X 0,Y 397.071,Z 344.653,A -85,B 0,C 180,E1 -11102.07,E2 -11102.07} C_VEL
LIN {X 0,Y 397.111,Z 344.646,A -85,B 0,C 180,E1 -11105.501,E2 -11105.501} C_VEL
LIN {X 0,Y 397.084,Z 344.649,A -85,B 0,C 180,E1 -11108.853,E2 -11108.853} C_VEL
LIN {X 0,Y 397.045,Z 344.651,A -85,B 0,C 180,E1 -11112.268,E2 -11112.268} C_VEL
LIN {X 0,Y 397.076,Z 344.65,A -85,B 0,C 180,E1 -11115.068,E2 -11115.068} C_VEL
LIN {X 0,Y 397.042,Z 344.65,A -85,B 0,C 180,E1 -11118.022,E2 -11118.022} C_VEL
LIN {X 0,Y 397.081,Z 344.637,A -85,B 0,C 180,E1 -11121.722,E2 -11121.722} C_VEL
LIN {X 0,Y 397.108,Z 344.64,A -85,B 0,C 180,E1 -11125.505,E2 -11125.505} C_VEL
LIN {X 0,Y 397.064,Z 344.65,A -85,B 0,C 180,E1 -11129.116,E2 -11129.116} C_VEL
LIN {X 0,Y 397.05,Z 344.647,A -85,B 0,C 180,E1 -11132.25,E2 -11132.25} C_VEL
LIN {X 0,Y 397.089,Z 344.638,A -85,B 0,C 180,E1 -11134.864,E2 -11134.864} C_VEL
LIN {X 0,Y 397.081,Z 344.646,A -85,B 0,C 180,E1 -11138.18,E2 -11138.18} C_VEL
LIN {X 0,Y 397.143,Z 344.625,A -85,B 0,C 180,E1 -11141.425,E2 -11141.425} C_VEL
LIN {X 0,Y 397.16,Z 344.64,A -85,B 0,C 180,E1 -11144.607,E2 -11144.607} C_VEL
LIN {X 0,Y 397.203,Z 344.628,A -85,B 0,C 180,E1 -11147.741,E2 -11147.741} C_VEL
LIN {X 0,Y 397.22,Z 344.627,A -85,B 0,C 180,E1 -11150.837,E2 -11150.837} C_VEL
LIN {X 0,Y 397.3,Z 344.618,A -85,B 0,C 180,E1 -11153.907,E2 -11153.907} C_VEL
LIN {X 0,Y 397.428,Z 344.603,A -85,B 0,C 180,E1 -11157.973,E2 -11157.973} C_VEL
LIN {X 0,Y 397.425,Z 344.604,A -85,B 0,C 180,E1 -11162.027,E2 -11162.027} C_VEL
LIN {X 0,Y 397.315,Z 344.617,A -85,B 0,C 180,E1 -11166.092,E2 -11166.092} C_VEL
LIN {X 0,Y 397.211,Z 344.628,A -85,B 0,C 180,E1 -11169.163,E2 -11169.163} C_VEL
LIN {X 0,Y 397.198,Z 344.632,A -85,B 0,C 180,E1 -11172.259,E2 -11172.259} C_VEL
LIN {X 0,Y 397.163,Z 344.634,A -85,B 0,C 180,E1 -11175.393,E2 -11175.393} C_VEL
LIN {X 0,Y 397.142,Z 344.642,A -85,B 0,C 180,E1 -11178.574,E2 -11178.574} C_VEL
LIN {X 0,Y 397.08,Z 344.635,A -85,B 0,C 180,E1 -11181.819,E2 -11181.819} C_VEL
LIN {X 0,Y 397.089,Z 344.644,A -85,B 0,C 180,E1 -11185.136,E2 -11185.136} C_VEL
LIN {X 0,Y 397.051,Z 344.639,A -85,B 0,C 180,E1 -11188.549,E2 -11188.549} C_VEL
LIN {X 0,Y 397.067,Z 344.649,A -85,B 0,C 180,E1 -11191.837,E2 -11191.837} C_VEL
LIN {X 0,Y 397.104,Z 344.647,A -85,B 0,C 180,E1 -11194.495,E2 -11194.495} C_VEL
LIN {X 0,Y 397.076,Z 344.649,A -85,B 0,C 180,E1 -11198.278,E2 -11198.278} C_VEL
LIN {X 0,Y 397.038,Z 344.653,A -85,B 0,C 180,E1 -11201.977,E2 -11201.977} C_VEL
LIN {X 0,Y 397.073,Z 344.648,A -85,B 0,C 180,E1 -11205.071,E2 -11205.071} C_VEL
LIN {X 0,Y 397.04,Z 344.657,A -85,B 0,C 180,E1 -11208.025,E2 -11208.025} C_VEL
LIN {X 0,Y 397.077,Z 344.65,A -85,B 0,C 180,E1 -11211.725,E2 -11211.725} C_VEL
LIN {X 0,Y 397.108,Z 344.646,A -85,B 0,C 180,E1 -11215.507,E2 -11215.507} C_VEL
LIN {X 0,Y 397.068,Z 344.648,A -85,B 0,C 180,E1 -11219.119,E2 -11219.119} C_VEL
LIN {X 0,Y 397.099,Z 344.668,A -85,B 0,C 180,E1 -11219.884,E2 -11219.884} C_VEL
LIN {X 0,Y 399.99,Z 357.314,A -85,B 0,C 180,E1 -11222.819,E2 -11222.819} C_VEL
LIN {X 0,Y 401.764,Z 366.705,A -85,B 0,C 180,E1 -11224.902,E2 -11224.902} C_VEL
LIN {X 0,Y 401.404,Z 370.451,A -85,B 0,C 180,E1 -11225.652,E2 -11225.652} C_VEL
LIN {X 0,Y 406.91,Z 398.385,A -85,B 0,C 180,E1 -11226.54,E2 -11226.54} C_VEL
LIN {X 0,Y 407.401,Z 401.332,A -85,B 0,C 180,E1 -11226.626,E2 -11226.626} C_VEL
LIN {X 0,Y 405.607,Z 507.469,A -85,B 0,C 180,E1 -11228.531,E2 -11228.531} C_VEL
LIN {X 0,Y 404.97,Z 521.569,A -85,B 0,C 180,E1 -11228.962,E2 -11228.962} C_VEL
LIN {X 0,Y 404.144,Z 535.258,A -85,B 0,C 180,E1 -11229.583,E2 -11229.583} C_VEL
LIN {X 0,Y 403.292,Z 547.195,A -85,B 0,C 180,E1 -11230.3,E2 -11230.3} C_VEL
LIN {X 0,Y 402.234,Z 559.925,A -85,B 0,C 180,E1 -11231.275,E2 -11231.275} C_VEL
LIN {X 0,Y 401.053,Z 571.809,A -85,B 0,C 180,E1 -11232.407,E2 -11232.407} C_VEL
LIN {X 0,Y 399.92,Z 582.666,A -85,B 0,C 180,E1 -11233.671,E2 -11233.671} C_VEL
LIN {X 0,Y 398.763,Z 593.397,A -85,B 0,C 180,E1 -11235.195,E2 -11235.195} C_VEL
LIN {X 0,Y 397.906,Z 602.257,A -85,B 0,C 180,E1 -11236.727,E2 -11236.727} C_VEL
LIN {X 0,Y 397.248,Z 609.63,A -85,B 0,C 180,E1 -11238.263,E2 -11238.263} C_VEL
LIN {X 0,Y 396.635,Z 615.774,A -85,B 0,C 180,E1 -11239.796,E2 -11239.796} C_VEL
LIN {X 0,Y 396.147,Z 622.301,A -85,B 0,C 180,E1 -11241.842,E2 -11241.842} C_VEL
LIN {X 0,Y 395.908,Z 627.191,A -85,B 0,C 180,E1 -11243.887,E2 -11243.887} C_VEL
LIN {X 0,Y 395.755,Z 630.587,A -85,B 0,C 180,E1 -11245.928,E2 -11245.928} C_VEL
LIN {X 0,Y 395.716,Z 632.592,A -85,B 0,C 180,E1 -11247.966,E2 -11247.966} C_VEL
LIN {X 0,Y 395.758,Z 633.254,A -85,B 0,C 180,E1 -11250.002,E2 -11250.002} C_VEL
LIN {X 0,Y 395.717,Z 632.583,A -85,B 0,C 180,E1 -11252.037,E2 -11252.037} C_VEL
LIN {X 0,Y 395.754,Z 630.569,A -85,B 0,C 180,E1 -11254.075,E2 -11254.075} C_VEL
LIN {X 0,Y 395.91,Z 627.167,A -85,B 0,C 180,E1 -11256.116,E2 -11256.116} C_VEL
LIN {X 0,Y 396.15,Z 622.275,A -85,B 0,C 180,E1 -11258.161,E2 -11258.161} C_VEL
LIN {X 0,Y 396.639,Z 615.74,A -85,B 0,C 180,E1 -11260.207,E2 -11260.207} C_VEL
LIN {X 0,Y 397.344,Z 608.467,A -85,B 0,C 180,E1 -11261.996,E2 -11261.996} C_VEL
LIN {X 0,Y 398.119,Z 600.055,A -85,B 0,C 180,E1 -11263.68,E2 -11263.68} C_VEL
LIN {X 0,Y 399.137,Z 590.008,A -85,B 0,C 180,E1 -11265.316,E2 -11265.316} C_VEL
